FUNCTION_BLOCK "LMQTT_Client"
{ S7_Optimized_Access := 'TRUE' }
AUTHOR : 'Siemens Industry Online Support'
FAMILY : LMQTT
VERSION : 4.0
   VAR_INPUT
      enable : Bool;
      publish : Bool;
      subscribe : Bool;
      unsubscribe : Bool;
      qos : USInt;
      "retain" : Bool;
      publishMsgLen : UDInt := 0;
      willMsgLen : UInt := 0;
      timeOut { S7_HiddenAssignment := 'HideIfNoParamAssigned'} : Time := T#5s;
   END_VAR

   VAR_OUTPUT
      valid { ExternalWritable := 'False'} : Bool;
      done { ExternalWritable := 'False'} : Bool;
      busy { ExternalWritable := 'False'} : Bool;
      error { ExternalWritable := 'False'} : Bool;
      status { ExternalWritable := 'False'} : Word := #STATUS_NO_CALL;
      diagnostics { ExternalWritable := 'False'} : "typeDiagnostics";
      receivedMsgStatus { ExternalWritable := 'False'} : USInt;
      receivedMsgDataLen { ExternalWritable := 'False'} : UDInt;
   END_VAR

   VAR_IN_OUT
      connParam : "LMQTT_typeConnParam";
      clientIdentifier : WString;
      username : WString;
      password : WString;
      willtopic : WString;
      willMsgPayload : Array[*] of Byte;
      mqttTopic : WString;
      publishMsgPayload : Array[*] of Byte;
      receivedTopic : WString;
      receivedMsgPayload : Array[*] of Byte;
   END_VAR

   VAR
      statEnableOld { ExternalAccessible := 'False'; ExternalVisible := 'False'; ExternalWritable := 'False'} : Bool;
      statValid { ExternalAccessible := 'False'; ExternalVisible := 'False'; ExternalWritable := 'False'} : Bool;
      statBusy { ExternalAccessible := 'False'; ExternalVisible := 'False'; ExternalWritable := 'False'} : Bool;
      statError { ExternalAccessible := 'False'; ExternalVisible := 'False'; ExternalWritable := 'False'} : Bool;
      statErrorUserCleared { ExternalAccessible := 'False'; ExternalVisible := 'False'; ExternalWritable := 'False'} : Bool;
      statErrorAutoCleared { ExternalAccessible := 'False'; ExternalVisible := 'False'; ExternalWritable := 'False'} : Bool;
      statStatus { ExternalAccessible := 'False'; ExternalVisible := 'False'; ExternalWritable := 'False'} : Word := #STATUS_NO_CALL;
      statDone { ExternalAccessible := 'False'; ExternalVisible := 'False'; ExternalWritable := 'False'} : Bool;
      statRcvMsgStatus { ExternalAccessible := 'False'; ExternalVisible := 'False'; ExternalWritable := 'False'} : USInt;
      statRcvMsgDataLen { ExternalAccessible := 'False'; ExternalVisible := 'False'; ExternalWritable := 'False'} : UDInt;
      statSubfunctionStatus { ExternalAccessible := 'False'; ExternalVisible := 'False'; ExternalWritable := 'False'} : Word;
      statFBErrorState { ExternalAccessible := 'False'; ExternalVisible := 'False'; ExternalWritable := 'False'} : DInt;
      statFBState { ExternalAccessible := 'False'; ExternalVisible := 'False'; ExternalWritable := 'False'} : DInt := #FB_STATE_NO_PROCESSING;
      statMqttConnectState { ExternalAccessible := 'False'; ExternalVisible := 'False'; ExternalWritable := 'False'} : DInt := #MQTT_CONNECT_STATE_NO_PROCESSING;
      statMqttCommandState { ExternalAccessible := 'False'; ExternalVisible := 'False'; ExternalWritable := 'False'} : DInt := #MQTT_COMMAND_STATE_NO_PROCESSING;
      statDisablingCompleted { ExternalAccessible := 'False'; ExternalVisible := 'False'; ExternalWritable := 'False'} : Bool;
      statEmptyDiagnostics { ExternalAccessible := 'False'; ExternalVisible := 'False'; ExternalWritable := 'False'; S7_SetPoint := 'False'} : "typeDiagnostics";
      statConnParam { ExternalAccessible := 'False'; ExternalVisible := 'False'; ExternalWritable := 'False'} : Struct
         isQDN { ExternalAccessible := 'False'; ExternalVisible := 'False'; ExternalWritable := 'False'} : Bool;
         paramQDN {InstructionName := 'TCON_QDN_SEC'; LibVersion := '1.0'; ExternalAccessible := 'False'; ExternalVisible := 'False'; ExternalWritable := 'False'; S7_SetPoint := 'False'} : TCON_QDN_SEC;
         paramIP {InstructionName := 'TCON_IP_V4_SEC'; LibVersion := '1.0'; ExternalAccessible := 'False'; ExternalVisible := 'False'; ExternalWritable := 'False'; S7_SetPoint := 'False'} : TCON_IP_V4_SEC;
      END_STRUCT;
      instTsendC {InstructionName := 'TSEND_C'; LibVersion := '3.2'; ExternalAccessible := 'False'; ExternalVisible := 'False'; ExternalWritable := 'False'; S7_SetPoint := 'False'} : TSEND_C;
      instTrcv {InstructionName := 'TRCV'; LibVersion := '4.0'; ExternalAccessible := 'False'; ExternalVisible := 'False'; ExternalWritable := 'False'; S7_SetPoint := 'False'} : TRCV;
      statSendBuffer { ExternalAccessible := 'False'; ExternalVisible := 'False'; ExternalWritable := 'False'} : Array[0..#MAX_BUFFER_LEN_SEND] of Byte;
      statRcvBuffer { ExternalAccessible := 'False'; ExternalVisible := 'False'; ExternalWritable := 'False'} : Array[0..#MAX_BUFFER_LEN_RCV] of Byte;
      statPublishOld { ExternalAccessible := 'False'; ExternalVisible := 'False'; ExternalWritable := 'False'} : Bool;
      statSubscribeOld { ExternalAccessible := 'False'; ExternalVisible := 'False'; ExternalWritable := 'False'} : Bool;
      statUnsubscribeOld { ExternalAccessible := 'False'; ExternalVisible := 'False'; ExternalWritable := 'False'} : Bool;
      statTsendcReq { ExternalAccessible := 'False'; ExternalVisible := 'False'; ExternalWritable := 'False'} : Bool;
      statTsendcEnable { ExternalAccessible := 'False'; ExternalVisible := 'False'; ExternalWritable := 'False'} : Bool;
      statTsendcLen { ExternalAccessible := 'False'; ExternalVisible := 'False'; ExternalWritable := 'False'} : UDInt;
      statEnableTimerCommandWatchdog { ExternalAccessible := 'False'; ExternalVisible := 'False'; ExternalWritable := 'False'} : Bool;
      instTimerCommandWatchdog {InstructionName := 'IEC_TIMER'; LibVersion := '1.0'; ExternalAccessible := 'False'; ExternalVisible := 'False'; ExternalWritable := 'False'; S7_SetPoint := 'False'} : IEC_TIMER;
      statEnableMqttKeepAliveTimer { ExternalAccessible := 'False'; ExternalVisible := 'False'; ExternalWritable := 'False'} : Bool;
      statMqttKeepAliveUsed { ExternalAccessible := 'False'; ExternalVisible := 'False'; ExternalWritable := 'False'} : Bool;
      statMqttKeepAliveTime { ExternalAccessible := 'False'; ExternalVisible := 'False'; ExternalWritable := 'False'} : Time;
      instMqttKeepAliveTimer {InstructionName := 'IEC_TIMER'; LibVersion := '1.0'; ExternalAccessible := 'False'; ExternalVisible := 'False'; ExternalWritable := 'False'; S7_SetPoint := 'False'} : IEC_TIMER;
      statSendBufferPos { ExternalAccessible := 'False'; ExternalVisible := 'False'; ExternalWritable := 'False'} : UInt;
      statPaketHeaderEncodeDone { ExternalAccessible := 'False'; ExternalVisible := 'False'; ExternalWritable := 'False'} : Bool;
      statSendPaketTotalRemLen { ExternalAccessible := 'False'; ExternalVisible := 'False'; ExternalWritable := 'False'} : UDInt;
      statEncodedRemPaketLenAsByte { ExternalAccessible := 'False'; ExternalVisible := 'False'; ExternalWritable := 'False'} : Byte;
      statUsernameLenUtf8Encoded { ExternalAccessible := 'False'; ExternalVisible := 'False'; ExternalWritable := 'False'} : UInt;
      statPasswordLenUtf8Encoded { ExternalAccessible := 'False'; ExternalVisible := 'False'; ExternalWritable := 'False'} : UInt;
      statWillTopicLenUtf8Encoded { ExternalAccessible := 'False'; ExternalVisible := 'False'; ExternalWritable := 'False'} : UInt;
      statClientIdLenUtf8Encoded { ExternalAccessible := 'False'; ExternalVisible := 'False'; ExternalWritable := 'False'} : UInt;
      statWillQos { ExternalAccessible := 'False'; ExternalVisible := 'False'; ExternalWritable := 'False'} : USInt;
      statWillRetain { ExternalAccessible := 'False'; ExternalVisible := 'False'; ExternalWritable := 'False'} : Bool;
      statWillMessageCnt { ExternalAccessible := 'False'; ExternalVisible := 'False'; ExternalWritable := 'False'} : UInt;
      statClientIdPos { ExternalAccessible := 'False'; ExternalVisible := 'False'; ExternalWritable := 'False'} : DInt;
      statClientIdEncodeState { ExternalAccessible := 'False'; ExternalVisible := 'False'; ExternalWritable := 'False'} : DInt;
      statWillMessagePos { ExternalAccessible := 'False'; ExternalVisible := 'False'; ExternalWritable := 'False'} : DInt;
      statWillMessageEncodeState { ExternalAccessible := 'False'; ExternalVisible := 'False'; ExternalWritable := 'False'} : DInt;
      statWillTopicPos { ExternalAccessible := 'False'; ExternalVisible := 'False'; ExternalWritable := 'False'} : DInt;
      statWillTopicEncodeState { ExternalAccessible := 'False'; ExternalVisible := 'False'; ExternalWritable := 'False'} : DInt;
      statUserNamePos { ExternalAccessible := 'False'; ExternalVisible := 'False'; ExternalWritable := 'False'} : DInt;
      statUserNameEncodeState { ExternalAccessible := 'False'; ExternalVisible := 'False'; ExternalWritable := 'False'} : DInt;
      statPasswordPos { ExternalAccessible := 'False'; ExternalVisible := 'False'; ExternalWritable := 'False'} : DInt;
      statPasswordEncodeState { ExternalAccessible := 'False'; ExternalVisible := 'False'; ExternalWritable := 'False'} : DInt;
      statPaketId { ExternalAccessible := 'False'; ExternalVisible := 'False'; ExternalWritable := 'False'} : UInt;
      statPublishTopicLenUtf8Encoded { ExternalAccessible := 'False'; ExternalVisible := 'False'; ExternalWritable := 'False'} : UInt;
      statPublishQos { ExternalAccessible := 'False'; ExternalVisible := 'False'; ExternalWritable := 'False'} : USInt;
      statPublishMessageCnt { ExternalAccessible := 'False'; ExternalVisible := 'False'; ExternalWritable := 'False'} : UDInt;
      statPublishTopicEncodeState { ExternalAccessible := 'False'; ExternalVisible := 'False'; ExternalWritable := 'False'} : DInt;
      statPublishTopicPos { ExternalAccessible := 'False'; ExternalVisible := 'False'; ExternalWritable := 'False'} : DInt;
      statPaketIdEncoded { ExternalAccessible := 'False'; ExternalVisible := 'False'; ExternalWritable := 'False'} : Bool;
      statPublishEncodeMessageState { ExternalAccessible := 'False'; ExternalVisible := 'False'; ExternalWritable := 'False'} : DInt;
      statPublishMessagePos { ExternalAccessible := 'False'; ExternalVisible := 'False'; ExternalWritable := 'False'} : DInt;
      statSubscribeQos { ExternalAccessible := 'False'; ExternalVisible := 'False'; ExternalWritable := 'False'} : USInt;
      statSubscribeQosEncoded { ExternalAccessible := 'False'; ExternalVisible := 'False'; ExternalWritable := 'False'} : Bool;
      statSubscribeTopicPos { ExternalAccessible := 'False'; ExternalVisible := 'False'; ExternalWritable := 'False'} : DInt;
      statSubscribeTopicEncodeState { ExternalAccessible := 'False'; ExternalVisible := 'False'; ExternalWritable := 'False'} : DInt;
      statSubscribeTopicLenUtf8Encoded { ExternalAccessible := 'False'; ExternalVisible := 'False'; ExternalWritable := 'False'} : UInt;
      statUnsubscribeTopicPos { ExternalAccessible := 'False'; ExternalVisible := 'False'; ExternalWritable := 'False'} : DInt;
      statUnsubscribeTopicEncodeState { ExternalAccessible := 'False'; ExternalVisible := 'False'; ExternalWritable := 'False'} : DInt;
      statUnsubscribeTopicLenUtf8Encoded { ExternalAccessible := 'False'; ExternalVisible := 'False'; ExternalWritable := 'False'} : UInt;
      statRcvMsgQoS { ExternalAccessible := 'False'; ExternalVisible := 'False'; ExternalWritable := 'False'} : UInt;
      statRcvMsgTotalLen { ExternalAccessible := 'False'; ExternalVisible := 'False'; ExternalWritable := 'False'} : UDInt;
      statRcvMsgTopicLen { ExternalAccessible := 'False'; ExternalVisible := 'False'; ExternalWritable := 'False'} : UInt;
      statRcvMsgPayloadLen { ExternalAccessible := 'False'; ExternalVisible := 'False'; ExternalWritable := 'False'} : UDInt;
      statRcvMsgPaketId { ExternalAccessible := 'False'; ExternalVisible := 'False'; ExternalWritable := 'False'} : Word;
      statRcvMsgTopicPos { ExternalAccessible := 'False'; ExternalVisible := 'False'; ExternalWritable := 'False'} : DInt;
      statRcvMsgPayloadPos { ExternalAccessible := 'False'; ExternalVisible := 'False'; ExternalWritable := 'False'} : DInt;
      statRcvMsgDecodeState { ExternalAccessible := 'False'; ExternalVisible := 'False'; ExternalWritable := 'False'} : DInt;
      statRcvMsgInternalStatus { ExternalAccessible := 'False'; ExternalVisible := 'False'; ExternalWritable := 'False'} : USInt;
      statMqttPubRecRcv { ExternalAccessible := 'False'; ExternalVisible := 'False'; ExternalWritable := 'False'} : USInt;
      statSendPubAckMsg { ExternalAccessible := 'False'; ExternalVisible := 'False'; ExternalWritable := 'False'} : Bool;
      statPubRecReady { ExternalAccessible := 'False'; ExternalVisible := 'False'; ExternalWritable := 'False'} : Bool;
      statCommandInputOld { ExternalAccessible := 'False'; ExternalVisible := 'False'; ExternalWritable := 'False'} : Bool;
      statCommandInputBackup { ExternalAccessible := 'False'; ExternalVisible := 'False'; ExternalWritable := 'False'} : Byte;
   END_VAR

   VAR_TEMP
      tempEnable : Bool;
      tempSubscribe : Bool;
      tempPublish : Bool;
      tempUnsubscribe : Bool;
      tempTsendcDone : Bool;
      tempTsendcBusy : Bool;
      tempTsendcError : Bool;
      tempTsendcStatus : Word;
      tempTrcvNdr : Bool;
      tempTrcvBusy : Bool;
      tempTrcvError : Bool;
      tempTrcvStatus : Word;
      tempTrcvRcvdLen : UDInt;
      tempTrcvBufferPos : DInt;
      tempUserFlag : Bool;
      tempPasswordFlag : Bool;
      tempWillFlag : Bool;
      tempWillQoS1 : Bool;
      tempWillQoS2 : Bool;
      tempMaxWillMsgLen : DInt;
      tempLowerWillMsgArrayBoundary : DInt;
      tempLoopCounter : DInt;
      tempBytesUsedUtf8 : USInt;
      tempErrorConvertUtf8 : Bool;
      tempStatusConvertUtf8 : Word;
      tempConvertedUtf8 : DWord;
      tempWordForSliceAddress : Word;
      tempCommandInput : Byte;
      tempRcvMsgTypeCase : Byte;
      tempMaxPublishDataArrayLen : DInt;
      tempMqttConnAckRcvStatus : USInt;
      tempMqttPingRspRcv : USInt;
      tempMqttPubAckRcv : USInt;
      tempMqttPubCompRcv : USInt;
      tempMqttSubAckRcv : USInt;
      tempMqttUnSubAckRcv : USInt;
      tempLowerBoundPublishDataArray : DInt;
      tempMultiplierToDecode : UDInt;
      tempReceivedTopicStringMaxLen : DInt;
      tempReceivedMsgDataArrayTotalLen : DInt;
      tempUpperBoundRcvMsgDataArray : DInt;
      tempFirstChar : Int;
   END_VAR

   VAR CONSTANT
      FB_STATE_NO_PROCESSING : DInt := 0;
      FB_STATE_VALIDATE_INPUT : DInt := 10;
      FB_STATE_TCP_CONNECTING : DInt := 20;
      FB_STATE_OPERATING_MONITOR_TCP : DInt := 30;
      FB_STATE_TCP_RECONNECTING : DInt := 40;
      FB_STATE_DISABLING : DInt := 90;
      MQTT_CONNECT_STATE_NO_PROCESSING : DInt := 0;
      MQTT_CONNECT_STATE_BUILD_PAKET : DInt := 100;
      MQTT_CONNECT_STATE_SEND_PAKET_WAIT_FOR_CONNACK : DInt := 200;
      MQTT_CONNECT_STATE_CONNECTED : DInt := 300;
      MQTT_CONNECT_STATE_DISCONNECTED : DInt := 400;
      MQTT_COMMAND_STATE_NO_PROCESSING : DInt := 0;
      MQTT_COMMAND_STATE_BUILD_PUBLISH : DInt := 1;
      MQTT_COMMAND_STATE_SEND_PUBLISH : DInt := 1000;
      MQTT_COMMAND_STATE_BUILD_SUBSCRIBE : DInt := 2;
      MQTT_COMMAND_STATE_SEND_SUBSCRIBE : DInt := 2000;
      MQTT_COMMAND_STATE_BUILD_UNSUBSCRIBE : DInt := 4;
      MQTT_COMMAND_STATE_SEND_UNSUBSCRIBE : DInt := 3000;
      MQTT_COMMAND_STATE_SEND_PING : DInt := 8000;
      MQTT_COMMAND_STATE_PING_RESP : DInt := 9000;
      STATUS_JOB_EXECUTED : Word := 16#0000;
      STATUS_NO_CALL : Word := 16#7000;
      STATUS_FIRST_CALL : Word := 16#7001;
      STATUS_SUBSEQUENT_CALL : Word := 16#7002;
      STATUS_MQTT_CONNECTING : Word := 16#7003;
      STATUS_MQTT_CONNECTED : Word := 16#7004;
      STATUS_MQTT_PING : Word := 16#7005;
      STATUS_MQTT_PUBLISH : Word := 16#7006;
      STATUS_MQTT_SUBSCRIBE : Word := 16#7008;
      STATUS_MQTT_UNSUBSCRIBE : Word := 16#7010;
      ERR_UNDEFINED_STATE : Word := 16#8600;
      ERR_TCP_RECONNECTING : Word := 16#9000;
      ERR_CLIENT_ID_NULL : Word := 16#8200;
      ERR_BROKER_INVALID : Word := 16#8201;
      ERR_CNT_EXCEEDS_ARRAY_DIMENSION : Word := 16#8210;
      ERR_KEEPALIVE_INVALID : Word := 16#8220;
      ERR_QOS_INVALID : Word := 16#8230;
      ERR_TCON_FAILED : Word := 16#8601;
      ERR_TCON_TIMEOUT : Word := 16#8620;
      ERR_MQTT_REM_LEN_INVALID : Word := 16#8700;
      ERR_MQTT_MALFORMED_QOS_RECEIVED : Word := 16#8710;
      ERR_MQTT_CONNACK_INVALID_SESSION_FLAG : Word := 16#8720;
      ERR_MQTT_CONNACK_RETURN_CODE_INVALID : Word := 16#8730;
      ERR_MQTT_PAKET_ID_INVALID : Word := 16#8740;
      ERR_MQTT_SUBACK_FAILURE : Word := 16#8750;
      ERR_MQTT_COMMAND_MULTIPLE_INPUT : Word := 16#8001;
      ERR_MQTT_COMMAND_PUBLISH_TOPIC_INVALID : Word := 16#8300;
      ERR_MQTT_COMMAND_SUBSCRIBE_TOPIC_INVALID : Word := 16#8310;
      ERR_MQTT_COMMAND_UNSUBSCRIBE_TOPIC_INVALID : Word := 16#8320;
      ERR_MQTT_COMMAND_SEND_TIMEOUT : Word := 16#8650;
      ERR_MQTT_CONNECT_TIMEOUT : Word := 16#8670;
      MAX_BUFFER_LEN_RCV : UInt := 1459;
      MAX_BUFFER_LEN_SEND : UInt := 8191;
      EMPTY_BYTE : Byte := 16#00;
      NO_COMMAND : Byte := 16#00;
      EMPTY_STRING : String;
      EMPTY_WSTRING : WString;
      LEN_NULL : Int := 0;
      INIT_UDINT_1 : UDInt := 1;
      ARRAY_LEN_OFFSET_PLUS_1 : DInt := 1;
      FIRST_CHARACTER : DInt := 1;
      ONE_DIMENSION : UDInt := 1;
      FIRST_ENCODING : DInt := 1;
      SUBSEQUENT_ENCODING : DInt := 2;
      ENCODE_DONE : DInt := 3;
      NOT_USED_NO_ENCODING : DInt := 5;
      MSG_DECODE_STATE_NO_PROCESSING : DInt := 0;
      MSG_DECODE_STATE_TOPIC : DInt := 1;
      MSG_DECODE_STATE_PAKET_ID_MSB : DInt := 2;
      MSG_DECODE_STATE_PAKET_ID_LSB : DInt := 3;
      MSG_DECODE_STATE_PAYLOAD : DInt := 4;
      MSG_DECODE_STATUS_NO_NEW_MSG : USInt := 0;
      MSG_DECODE_STATUS_NEW_MSG_OK : USInt := 1;
      MSG_DECODE_STATUS_TOPIC_TOO_LONG : USInt := 2;
      MSG_DECODE_STATUS_PAYLOAD_TOO_LONG : USInt := 2;
      MQTT_QOS_0 : UInt := 0;
      MQTT_QOS_1 : UInt := 1;
      MQTT_QOS_2 : UInt := 2;
      REMAINING_LEN_3 : Byte := 16#03;
      REMAINING_LEN_2 : Byte := 16#02;
      REMAINIG_LEN_0 : Byte := 16#00;
      SUBSCRIBE_FAILURE : Byte := 16#80;
      MQTT_NO_SESSION_PRESENT : Byte := 16#00;
      KEEPALIVE_DISABLED : Time := t#0s;
      TSENDC_JOB_DONE : Word := 16#0000;
      TSENDC_COM_CLOSED : Word := 16#0003;
      TSENDC_EST_OK : Word := 16#7004;
      TSENDC_DISCONNECTED : Word := 16#7000;
      UINT_CONST_1000 : UInt := 1000;
      TWO_SECONDS : UInt := 2000;
      THREE_SECONDS : UInt := 3;
      UTF_1_BYTE_USED : USInt := 1;
      UTF_2_BYTE_USED : USInt := 2;
      UTF_3_BYTE_USED : USInt := 3;
      ONE_BYTE_LEN_INFO : UInt := 1;
      TWO_BYTE_LEN_INFO : UInt := 2;
      CONNECT_HEADER_10BYTE_LEN : UInt := 10;
      NO_RESPONSE : USInt := 0;
      RESPONSE_GOOD : USInt := 1;
      RESPONSE_PAKET_ID_INVALID : USInt := 2;
      RESPONSE_SUBSCRIBE_FAILED : USInt := 3;
      MQTT_MSG_TYPE_CONNECT : Byte := 16#10;
      MQTT_MSG_TYPE_CONNACK : Byte := 16#20;
      MQTT_MSG_TYPE_DISCONNECT : Byte := 16#E0;
      MQTT_MSG_TYPE_PUBLISH : Byte := 16#30;
      MQTT_MSG_TYPE_PUBACK : Byte := 16#40;
      MQTT_MSG_TYPE_PUBREC : Byte := 16#50;
      MQTT_MSG_TYPE_PUBREL : Byte := 16#62;
      MQTT_MSG_TYPE_PUBCOMP : Byte := 16#70;
      MQTT_MSG_TYPE_SUBSCRIBE : Byte := 16#82;
      MQTT_MSG_TYPE_UNSUBSCRIBE : Byte := 16#A2;
      MQTT_MSG_TYPE_SUBACK : Byte := 16#90;
      MQTT_MSG_TYPE_UNSUBACK : Byte := 16#B0;
      MQTT_MSG_TYPE_PING : Byte := 16#C0;
      MQTT_MSG_TYPE_PINGRESP : Byte := 16#D0;
      MQTT_MSG_TYPE_RCV_PUB_MESSAGE : Byte := 16#30;
      MQTT_MSG_TYPE_RCV_PUB_MESSAGE_QoS0 : Byte := 16#30;
      MQTT_MSG_TYPE_RCV_PUB_MESSAGE_QoS1 : Byte := 16#32;
      MQTT_MSG_TYPE_RCV_PUB_MESSAGE_QoS2 : Byte := 16#34;
      MQTT_MSG_TYPE_RCV_PUB_MESSAGE_BAD : Byte := 16#36;
      MQTT_MSG_DECODING : Byte := 16#FF;
      MQTT_CONNACK_ACCEPTED : Byte := 16#00;
      BIT_MASK_HIGHBITS : Byte := 16#F0;
      BIT_MASK_QOS : Byte := 16#F6;
      DEFAULT_VALUE_ZERO : Int := 0;
      SEND_LEN_MULTIPLIER_UDINT_128 : UDInt := 128;
      MAX_ALLOWED_PAKET_SIZE : UDInt := 2097152;
      DEFAULT_MULTIPLIER_BYTE_127 : Byte := 16#7F;
      CONN_PROTOCOL_NAME_0 : Byte := 16#00;
      CONN_PROTOCOL_NAME_4 : Byte := 16#04;
      CONN_PROTOCOL_MQTT_VERSION_3_1_1 : Byte := 16#04;
   END_VAR


BEGIN
	REGION BLOCK INFO HEADER
	  //===============================================================================
	  // SIEMENS (c)Copyright 2023
	  //-------------------------------------------------------------------------------
	  // Title:        LMQTT_Client
	  // Function:     This FB implements an MQTT client. A user can publish data and
	  //               subscribe to topics to receive data.
	  // Library:      LMQTT
	  // Author:       Siemens Industry Online Support
	  // Tested with:  CPU 1516-3 PN/DP FW 2.9
	  // Engineering:  TIA Portal V17
	  // Restrictions: --
	  // Requirements: S7-1200 with firmware V4.4 or higher
	  //               S7-1500 with firmware V2.0 or higher
	  //-------------------------------------------------------------------------------
	  // Change log table:
	  // Version  | Date       | Expert in charge       | Changes applied
	  //----------|------------|------------------------|------------------------------
	  // 04.00.03 | 2024-04-09 | Online Support         | Allowed lastWill without payload
	  // 04.00.03 | 2024-02-12 | Online Support         | Improved evaluation of broker address
	  // 04.00.02 | 2023-09-05 | Online Support         | Fixed bug that edge on publish/subscribe while PING is saved
	  // 04.00.01 | 2023-08-30 | Online Support         | Fixed bug at TRCV and ConnID
	  // 04.00.00 | 2023-08-04 | Online Support         | Broker can be addresses with hostname or IP address using one parameter
	  //                                                | Reordered interface
	  //                                                | Fixed bug at publish with QoS = 2
	  // 03.00.05 | 2023-02-23 | Online Support         | Fixed bug that in rare situations no new commands were accepted
	  // 03.00.04 | 2022-06-09 | Online Support         | Fixed bug that done was not set if input was reset
	  // 03.00.03 | 2021-05-07 | Online Support         | Minor bug fixes
	  // 03.00.00 | 2020-11-04 | Online Support         | New block interface with major improvements
	  // 02.02.02 | 2020-03-16 | Online Support         | Improved issue with validateSubjectAlternateNameOfServer not setting correct bit
	  // 02.02.01 | 2019-12-03 | Online Support         | Update to V16 and fusion with S7-1200 Lib
	  // 02.01.00 | 2019-11-10 | Online Support         | Minor connection improvements. Updated some comments
	  // 02.00.00 | 2018-06-04 | Online Support         | Added DNS support and Subscribe to topics
	  // 01.00.00 | 2017-06-06 | Online Support         | First released version
	  //===============================================================================
	END_REGION

	#tempEnable := #enable; // Work with temporary value / create process image
	#tempPublish := #publish;  // Work with temporary value / create process image - only checked when MQTT is connected
	#tempSubscribe := #subscribe;  // Work with temporary value / create process image - only checked when MQTT is connected
	#tempUnsubscribe := #unsubscribe;  // Work with temporary value / create process image - only checked when MQTT is connected


	REGION OUC_BLOCK_CALLS
	  //Only call if FB is processing
	  IF #statStatus <> #STATUS_NO_CALL THEN
	    // Connect and send
	    IF #statConnParam.isQDN = TRUE THEN // Call if host is a domain name
	      #instTsendC(REQ     := #statTsendcReq,
	                  CONT    := #statTsendcEnable,
	                  LEN     := #statTsendcLen,
	                  DONE    => #tempTsendcDone,
	                  BUSY    => #tempTsendcBusy,
	                  ERROR   => #tempTsendcError,
	                  STATUS  => #tempTsendcStatus,
	                  CONNECT := #statConnParam.paramQDN,
	                  DATA    := #statSendBuffer);

	    ELSE
	      #instTsendC(REQ     := #statTsendcReq,
	                  CONT    := #statTsendcEnable,
	                  LEN     := #statTsendcLen,
	                  DONE    => #tempTsendcDone,
	                  BUSY    => #tempTsendcBusy,
	                  ERROR   => #tempTsendcError,
	                  STATUS  => #tempTsendcStatus,
	                  CONNECT := #statConnParam.paramIP,
	                  DATA    := #statSendBuffer);
	    END_IF;

	    // Receive only when TCP operating
	    #instTrcv(EN_R     := (#statFBState = #FB_STATE_OPERATING_MONITOR_TCP),
	              ID       := #statConnParam.paramQDN.ConnPara.ID,
	              ADHOC    := true,
	              NDR      => #tempTrcvNdr,
	              BUSY     => #tempTrcvBusy,
	              ERROR    => #tempTrcvError,
	              STATUS   => #tempTrcvStatus,
	              RCVD_LEN => #tempTrcvRcvdLen,
	              DATA     := #statRcvBuffer);

	    //Monitor Time out
	    #instTimerCommandWatchdog.TON(IN := #statEnableTimerCommandWatchdog,
	                                  PT := #timeOut);
	    //Mqtt Keepalive Timer
	    #instMqttKeepAliveTimer.TON(IN := #statEnableMqttKeepAliveTimer,
	                                PT := #statMqttKeepAliveTime);
	  END_IF;
	END_REGION

	REGION ENABLING/DISABLING_FUNCTION_BLOCK
	  IF (#tempEnable = TRUE) AND (#statStatus = #STATUS_NO_CALL) THEN // Enable FB
	    // First call; initialize FB
	    #statValid := TRUE;
	    #statBusy := TRUE;
	    #statError := FALSE;
	    #statDone := FALSE;
	    #statErrorUserCleared := FALSE;
	    #statErrorAutoCleared := FALSE;
	    #statStatus := #STATUS_FIRST_CALL;
	    #statSubfunctionStatus := #STATUS_JOB_EXECUTED;
	    #statFBErrorState := 0;
	    #diagnostics := #statEmptyDiagnostics;
	    #statDisablingCompleted := FALSE;
	    // State machine - start functionality
	    #statFBState := #FB_STATE_VALIDATE_INPUT;

	    // Initialize functionality: reset of variables, diagnostics, etc.
	    #statPublishOld := FALSE;
	    #statSubscribeOld := FALSE;
	    #statUnsubscribeOld := FALSE;
	    #statConnParam.isQDN := FALSE;
	    #statTsendcReq := FALSE;
	    #statTsendcEnable := FALSE;
	    #statTsendcLen := 0;
	    #statEnableTimerCommandWatchdog := FALSE;
	    #statEnableMqttKeepAliveTimer := FALSE;
	    #statMqttKeepAliveTime := #KEEPALIVE_DISABLED;
	    #statMqttKeepAliveUsed := FALSE;
	    #statSendBufferPos := 0;
	    #statPaketHeaderEncodeDone := FALSE;
	    #statSendPaketTotalRemLen := 0;
	    #statEncodedRemPaketLenAsByte := #EMPTY_BYTE;
	    #statClientIdPos := 0;
	    #statClientIdEncodeState := 0;
	    #statClientIdLenUtf8Encoded := 0;
	    #statUserNamePos := 0;
	    #statUserNameEncodeState := #FIRST_ENCODING;
	    #statUsernameLenUtf8Encoded := 0;
	    #statPasswordPos := 0;
	    #statPasswordEncodeState := #FIRST_ENCODING;
	    #statPasswordLenUtf8Encoded := 0;
	    #statWillQos := 0;
	    #statWillRetain := FALSE;
	    #statWillMessageCnt := 0;
	    #statWillMessagePos := 0;
	    #statWillMessageEncodeState := #FIRST_ENCODING;
	    #statWillTopicLenUtf8Encoded := 0;
	    #statWillTopicPos := 0;
	    #statWillTopicEncodeState := #FIRST_ENCODING;
	    #statPaketId := 0;
	    #statPublishTopicLenUtf8Encoded := 0;
	    #statPublishQos := 0;
	    #statPublishMessageCnt := 0;
	    #statPublishTopicEncodeState := #FIRST_ENCODING;
	    #statPublishTopicPos := 0;
	    #statPaketIdEncoded := FALSE;
	    #statPublishEncodeMessageState := #FIRST_ENCODING;
	    #statPublishMessagePos := 0;
	    #statSubscribeQos := 0;
	    #statSubscribeQosEncoded := FALSE;
	    #statSubscribeTopicPos := 0;
	    #statSubscribeTopicEncodeState := #FIRST_ENCODING;
	    #statSubscribeTopicLenUtf8Encoded := 0;
	    #statUnsubscribeTopicPos := 0;
	    #statUnsubscribeTopicEncodeState := #FIRST_ENCODING;
	    #statUnsubscribeTopicLenUtf8Encoded := 0;
	    #statRcvMsgQoS := 0;
	    #statRcvMsgTotalLen := 0;
	    #statRcvMsgTopicLen := 0;
	    #statRcvMsgPayloadLen := 0;
	    #statRcvMsgPaketId := 0;
	    #statRcvMsgTopicPos := 0;
	    #statRcvMsgPayloadPos := 0;
	    #statRcvMsgDecodeState := #MSG_DECODE_STATE_NO_PROCESSING;
	    #statRcvMsgInternalStatus := 0;
	    #statRcvMsgStatus := 0;
	    #statRcvMsgDataLen := 0;
	    #statSendPubAckMsg := FALSE;

	    // Initialize functionality: call subsidiary FBs with FALSE
	    FILL_BLK(IN    := #EMPTY_BYTE,
	             COUNT := #MAX_BUFFER_LEN_SEND,
	             OUT   => #statSendBuffer[0]);
	    FILL_BLK(IN    := #EMPTY_BYTE,
	             COUNT := #MAX_BUFFER_LEN_RCV,
	             OUT   => #statRcvBuffer[0]);
	    RESET_TIMER(#instTimerCommandWatchdog);
	    RESET_TIMER(#instMqttKeepAliveTimer);

	    // INIT SUB STATE MACHINES
	    #statMqttConnectState := #MQTT_CONNECT_STATE_NO_PROCESSING;
	    #statMqttCommandState := #MQTT_COMMAND_STATE_NO_PROCESSING;
	    #statRcvMsgDecodeState := #MSG_DECODE_STATE_NO_PROCESSING;

	  ELSIF (#tempEnable = FALSE) AND (#statEnableOld = TRUE) THEN // Disable FB
	    #statFBState := #FB_STATE_DISABLING;
	  ELSIF (#statStatus = #STATUS_FIRST_CALL) THEN // Set status identifier of subsequent call
	    #statStatus := #STATUS_SUBSEQUENT_CALL;
	  END_IF;

	  // Edge detection 'enable' input
	  #statEnableOld := #tempEnable;
	END_REGION ENABLING/DISABLING

	IF (#statStatus = #STATUS_NO_CALL) THEN // Nothing to do -> End here to reduce "system load"
	  RETURN;
	END_IF;

	REGION STATE_MACHINE_FUNCTION_BLOCK_TCP
	  CASE #statFBState OF // State machine of FB
	    #FB_STATE_NO_PROCESSING: // No processing active (Note: this state must always be present and left empty)
	      ;

	    #FB_STATE_VALIDATE_INPUT: // Enabling active
	      REGION EVALUATE CONNECTION PARAMETERS
	        // Determine if host is domain name or IP address
	        #statConnParam.isQDN := NOT "IsIPAddress"(address := #connParam.broker, ipAddress => #statConnParam.paramIP.ConnPara.RemoteAddress);

	        IF #statConnParam.isQDN THEN // Broker address is a hostname
	          IF #connParam.broker[LEN(#connParam.broker)] = '.' THEN
	            #statConnParam.paramQDN.ConnPara.RemoteQDN := #connParam.broker;
	          ELSE
	            #statConnParam.paramQDN.ConnPara.RemoteQDN := CONCAT(IN1 := #connParam.broker, IN2 := '.');
	          END_IF;

	          #statConnParam.paramQDN.ConnPara.InterfaceId := #connParam.hwId;
	          #statConnParam.paramQDN.ConnPara.ID := #connParam.connId;
	          #statConnParam.paramQDN.ConnPara.ActiveEstablished := TRUE;
	          #statConnParam.paramQDN.ConnPara.RemotePort := #connParam."port";
	        ELSE // Broker address is an IP address
	          #statConnParam.paramIP.ConnPara.InterfaceId := #connParam.hwId;
	          #statConnParam.paramIP.ConnPara.ID := #statConnParam.paramQDN.ConnPara.ID := #connParam.connId;
	          #statConnParam.paramIP.ConnPara.ActiveEstablished := TRUE;
	          #statConnParam.paramIP.ConnPara.RemotePort := #connParam."port";
	        END_IF;

	        IF #connParam.tls.enableTls THEN
	          IF #statConnParam.isQDN THEN
	            #statConnParam.paramQDN.ActivateSecureConn := TRUE;
	            #statConnParam.paramQDN.ExtTLSCapabilities.%X0 := #connParam.tls.validateServerIdentity;
	            #statConnParam.paramQDN.TLSServerCertRef := #connParam.tls.brokerCert;
	            #statConnParam.paramQDN.TLSClientCertRef := #connParam.tls.clientCert;
	          ELSE
	            #statConnParam.paramIP.ActivateSecureConn := TRUE;
	            #statConnParam.paramIP.ExtTLSCapabilities.%X0 := #connParam.tls.validateServerIdentity;
	            #statConnParam.paramIP.TLSServerCertRef := #connParam.tls.brokerCert;
	            #statConnParam.paramIP.TLSClientCertRef := #connParam.tls.clientCert;
	          END_IF;
	        END_IF;
	      END_REGION EVALUATE CONNECTION PARAMETERS

	      REGION FB_VALIDATE_INPUT
	        //Check Input variables:
	        #tempMaxWillMsgLen := ABS(UPPER_BOUND(ARR := #willMsgPayload, DIM := #ONE_DIMENSION) - LOWER_BOUND(ARR := #willMsgPayload, DIM := #ONE_DIMENSION)) + #ARRAY_LEN_OFFSET_PLUS_1;

	        //Check Client ID len Must be > 0
	        IF LEN(#clientIdentifier) <= #LEN_NULL THEN
	          #statStatus := #ERR_CLIENT_ID_NULL; // Set correct status that identifies error clearly
	          #statSubfunctionStatus := #ERR_CLIENT_ID_NULL; // Status or return value of called FBs, FCs and system blocks
	          #statFBErrorState := #statFBState; // Set error state number for diagnostic
	          #statErrorUserCleared := TRUE;
	          //verify Will next
	        ELSIF #tempMaxWillMsgLen < #willMsgLen THEN
	          #statStatus := #ERR_CNT_EXCEEDS_ARRAY_DIMENSION; // Set correct status that identifies error clearly
	          #statSubfunctionStatus := #ERR_CNT_EXCEEDS_ARRAY_DIMENSION; // Status or return value of called FBs, FCs and system blocks
	          #statFBErrorState := #statFBState; // Set error state number for diagnostic
	          #statErrorUserCleared := TRUE;
	          ///CHECK WILL QOS
	        ELSIF #qos > #MQTT_QOS_2 THEN
	          #statStatus := #ERR_QOS_INVALID; // Set correct status that identifies error clearly
	          #statSubfunctionStatus := #ERR_QOS_INVALID; // Status or return value of called FBs, FCs and system blocks
	          #statFBErrorState := #statFBState; // Set error state number for diagnostic
	          #statErrorUserCleared := TRUE;
	        ELSIF (#connParam.keepAlive < #THREE_SECONDS) // IF Set to 1 or 2 seconds..
	          AND (#connParam.keepAlive > 0)
	        THEN
	          #statStatus := #ERR_KEEPALIVE_INVALID; // Set correct status that identifies error clearly
	          #statSubfunctionStatus := #ERR_KEEPALIVE_INVALID; // Status or return value of called FBs, FCs and system blocks
	          #statFBErrorState := #statFBState; // Set error state number for diagnostic
	          #statErrorUserCleared := TRUE;
	        ELSE
	          //Set Params for connection
	          //Set Client Id
	          #statWillQos := #qos;
	          //set Retain
	          #statWillRetain := #retain;
	          // Will message cnt
	          #statWillMessageCnt := #willMsgLen;

	          //Keepalive
	          IF #connParam.keepAlive = 0 THEN
	            #statMqttKeepAliveUsed := FALSE;
	          ELSE
	            #statMqttKeepAliveUsed := TRUE;
	            //KeepAliveTImer is set to ((Keep Alive converted to seconds) - 2s)
	            #statMqttKeepAliveTime := UINT_TO_TIME((#connParam.keepAlive * #UINT_CONST_1000 - #TWO_SECONDS));
	          END_IF;

	          //rdy to enable TCON
	          #statTsendcEnable := TRUE;
	          #statEnableTimerCommandWatchdog := TRUE;
	          #statFBState := #FB_STATE_TCP_CONNECTING;
	        END_IF;
	      END_REGION FB_VALIDATE_INPUT

	    #FB_STATE_TCP_CONNECTING: //Wait for TCP to be established
	      REGION FB_TCP_CONNECTING
	        //Check process:
	        IF #tempTsendcError = TRUE THEN //when error:
	          #statTsendcEnable := FALSE; //disable TsendC
	          #statEnableTimerCommandWatchdog := FALSE;
	          #statStatus := #ERR_TCON_FAILED; // Set correct status that identifies error clearly
	          #statSubfunctionStatus := #tempTsendcStatus; // Status or return value of called FBs, FCs and system blocks
	          #statFBErrorState := #statFBState; // Set error state number for diagnostic
	          #statErrorUserCleared := TRUE;
	        ELSIF #tempTsendcStatus = #TSENDC_EST_OK THEN //when successfull:
	          //     Communication connection established.
	          #statEnableTimerCommandWatchdog := FALSE;
	          //Monitor Connection
	          #statFBState := #FB_STATE_OPERATING_MONITOR_TCP;
	          // Begin MQTT Connection
	          #statMqttConnectState := #MQTT_CONNECT_STATE_BUILD_PAKET;
	          //set status
	          #statStatus := #STATUS_MQTT_CONNECTING;
	        ELSIF #instTimerCommandWatchdog.Q THEN
	          #statTsendcEnable := FALSE; //disable TsendC
	          #statEnableTimerCommandWatchdog := FALSE;
	          #statStatus := #ERR_TCON_TIMEOUT; // Set correct status that identifies error clearly
	          #statSubfunctionStatus := #ERR_TCON_TIMEOUT; // Status or return value of called FBs, FCs and system blocks
	          #statFBErrorState := #statFBState; // Set error state number for diagnostic
	          #statErrorUserCleared := TRUE;
	        END_IF;
	      END_REGION FB_TCP_CONNECTING
	    #FB_STATE_OPERATING_MONITOR_TCP: // Processing active
	      REGION FB_OPERATING_MONITOR_TCP
	        //Reset Status on Msg Output - will be set when a new message is completly processed and ready at outputs.
	        #statRcvMsgStatus := #MSG_DECODE_STATUS_NO_NEW_MSG;
	        //Reset TsendC Req from last  cycle Request:

	        #statTsendcReq := FALSE;

	        //Monitor Connection - if disconnect occured:
	        IF ((#tempTsendcStatus > #TSENDC_COM_CLOSED AND #tempTsendcStatus < #TSENDC_EST_OK) //Status connection interupt
	          OR #tempTsendcError = TRUE) // Or error
	          AND #tempTrcvNdr = FALSE // And no new data (to see if broker send information why connection was interrupted)
	        THEN
	          REGION CONNECTION_INTERRUPTED
	            //Status reconnecting
	            //SET MQTT to no operation
	            #statMqttConnectState := #MQTT_CONNECT_STATE_NO_PROCESSING;
	            #statMqttCommandState := #MQTT_COMMAND_STATE_NO_PROCESSING;
	            #statRcvMsgDecodeState := #MSG_DECODE_STATE_NO_PROCESSING;
	            //Reset Pub ack
	            #statSendPubAckMsg := FALSE;
	            //reset Done bit if still set, regardless of input:
	            #statDone := FALSE;
	            //reset Watchdog
	            #statEnableTimerCommandWatchdog := FALSE;
	            // reset headerEncode
	            #statPaketHeaderEncodeDone := FALSE;
	            //set error  information
	            #statStatus := #ERR_TCP_RECONNECTING; // Set correct status that identifies error clearly
	            #statSubfunctionStatus := #tempTsendcStatus;// Status or return value of called FBs, FCs and system blocks
	            #statFBErrorState := #statFBState; // Set error state number for diagnostic
	            #statErrorAutoCleared := TRUE;
	            //Wait for reconect - next state
	            #statFBState := #FB_STATE_TCP_RECONNECTING;
	          END_REGION REGION CONNECTION_INTERRUPTED
	        ELSE
	          //Connection is OK
	          //Sending and receiving works
	          //Check Trcv Buffer for new Data
	          IF #tempTrcvNdr THEN
	            REGION TRCV_NEW_DATA
	              //Evaluate the TrcvBuffer, reset buffer pos to start
	              #tempTrcvBufferPos := 0;
	              // Parse the whole RCV Buffer
	              WHILE #tempTrcvBufferPos < (UDINT_TO_DINT(#tempTrcvRcvdLen)) DO
	                // Parse the whole RCV Buffer, check wether header or decoding
	                IF #statRcvMsgDecodeState = #MSG_DECODE_STATE_NO_PROCESSING THEN
	                  //If no decoding is in progress, look for new message header
	                  #tempRcvMsgTypeCase := #statRcvBuffer[#tempTrcvBufferPos] AND #BIT_MASK_HIGHBITS;
	                ELSE
	                  //decode is in progress, go directly to decoding
	                  #tempRcvMsgTypeCase := #MQTT_MSG_DECODING;
	                END_IF;

	                CASE #tempRcvMsgTypeCase OF
	                  #MQTT_MSG_TYPE_CONNACK:  // Statement section case 1
	                    REGION RECEIVED_CONACK_PACKET
	                      #tempTrcvBufferPos += 1;
	                      IF #statRcvBuffer[#tempTrcvBufferPos] = #REMAINING_LEN_2 //remainng Length must be 2;
	                      THEN //
	                        #tempTrcvBufferPos += 1;
	                        //byte one is 0000 000X where X is if Session was set // so depending on clean session or not  evaluate answer of server
	                        IF #statRcvBuffer[#tempTrcvBufferPos] = #MQTT_NO_SESSION_PRESENT THEN
	                          #tempTrcvBufferPos += 1;
	                          //VALID Answer, check code
	                          IF #statRcvBuffer[#tempTrcvBufferPos] = #MQTT_CONNACK_ACCEPTED
	                          THEN
	                            //All good
	                            #tempTrcvBufferPos += 1;
	                            #tempMqttConnAckRcvStatus := #RESPONSE_GOOD; //evaluate in MQTT StateMachine Below the response
	                          ELSE
	                            //NOT VALID CONNACK from server shows session has a bad return code
	                            #statStatus := #ERR_MQTT_CONNACK_RETURN_CODE_INVALID; // Set correct status that identifies error clearly
	                            #statSubfunctionStatus := #statRcvBuffer[#tempTrcvBufferPos]; // Status or return value of called FBs, FCs and system blocks
	                            #statFBErrorState := #statFBState; // Set error state number for diagnostic
	                            #statErrorUserCleared := TRUE;
	                            // Exit loop
	                            EXIT;
	                          END_IF;
	                        ELSE
	                          //NOT VALID, CONNACK from server shows session present
	                          #statStatus := #ERR_MQTT_CONNACK_INVALID_SESSION_FLAG; // Set correct status that identifies error clearly
	                          #statSubfunctionStatus := #ERR_MQTT_CONNACK_INVALID_SESSION_FLAG; // Status or return value of called FBs, FCs and system blocks
	                          #statFBErrorState := #statFBState; // Set error state number for diagnostic
	                          #statErrorUserCleared := TRUE;
	                          // Exit loop
	                          EXIT;
	                        END_IF;
	                      ELSE // We got a CONNACK paket, but remaining length was not 2 (Error)
	                        #statStatus := #ERR_MQTT_REM_LEN_INVALID; // Set correct status that identifies error clearly
	                        #statSubfunctionStatus := #ERR_MQTT_REM_LEN_INVALID; // Status or return value of called FBs, FCs and system blocks
	                        #statFBErrorState := #statFBState; // Set error state number for diagnostic
	                        #statErrorUserCleared := TRUE;
	                        // Exit loop
	                        EXIT;
	                      END_IF;
	                    END_REGION RECEIVED_CONACK_PACKET

	                  #MQTT_MSG_TYPE_PINGRESP:
	                    REGION RECEIVED_PINGRESP_PACKET
	                      #tempTrcvBufferPos += 1;
	                      IF #statRcvBuffer[#tempTrcvBufferPos] = #REMAINIG_LEN_0 //remainng Length must be 0;
	                      THEN
	                        #tempTrcvBufferPos += 1;
	                        #tempMqttPingRspRcv := #RESPONSE_GOOD; //evaluate in MQTT StateMachine Below the response
	                      ELSE// We got a Pingrsp paket, but remaining length was not 0 (Error)
	                        #statStatus := #ERR_MQTT_REM_LEN_INVALID; // Set correct status that identifies error clearly
	                        #statSubfunctionStatus := #ERR_MQTT_REM_LEN_INVALID; // Status or return value of called FBs, FCs and system blocks
	                        #statFBErrorState := #statFBState; // Set error state number for diagnostic
	                        #statErrorUserCleared := TRUE;
	                        // Exit loop
	                        EXIT;
	                      END_IF;
	                    END_REGION RECEIVED_PINGRESP_PAKET

	                  #MQTT_MSG_TYPE_PUBACK:
	                    REGION RECEIVED_PUBACK_PAKET
	                      #tempTrcvBufferPos += 1;
	                      IF #statRcvBuffer[#tempTrcvBufferPos] = #REMAINING_LEN_2 //remainng Length must be 2;
	                      THEN //
	                        #tempTrcvBufferPos += 1;
	                        #tempWordForSliceAddress := UINT_TO_WORD(#statPaketId);
	                        IF #statRcvBuffer[#tempTrcvBufferPos] = #tempWordForSliceAddress.%B1 THEN
	                          #tempTrcvBufferPos += 1;
	                          IF #statRcvBuffer[#tempTrcvBufferPos] = #tempWordForSliceAddress.%B0 THEN
	                            #tempTrcvBufferPos += 1;
	                            #tempMqttPubAckRcv := #RESPONSE_GOOD;
	                          ELSE
	                            #tempTrcvBufferPos += 1;
	                            #tempMqttPubAckRcv := #RESPONSE_PAKET_ID_INVALID;
	                          END_IF;
	                        ELSE
	                          #tempTrcvBufferPos += 1;
	                          #tempMqttPubAckRcv := #RESPONSE_PAKET_ID_INVALID;
	                        END_IF;
	                      ELSE
	                        #statStatus := #ERR_MQTT_REM_LEN_INVALID; // Set correct status that identifies error clearly
	                        #statSubfunctionStatus := #ERR_MQTT_REM_LEN_INVALID; // Status or return value of called FBs, FCs and system blocks
	                        #statFBErrorState := #statFBState; // Set error state number for diagnostic
	                        #statErrorUserCleared := TRUE;
	                        // Exit loop
	                        EXIT;
	                      END_IF;
	                    END_REGION RECEIVED_PUBACK_PAKET

	                  #MQTT_MSG_TYPE_PUBREC:
	                    REGION RECEIVED_PUBREC_PAKET
	                      #tempTrcvBufferPos += 1;
	                      IF #statRcvBuffer[#tempTrcvBufferPos] = #REMAINING_LEN_2 //remainng Length must be 2;
	                      THEN //
	                        #tempTrcvBufferPos += 1;
	                        #tempWordForSliceAddress := UINT_TO_WORD(#statPaketId);
	                        IF #statRcvBuffer[#tempTrcvBufferPos] = #tempWordForSliceAddress.%B1 THEN
	                          #tempTrcvBufferPos += 1;
	                          IF #statRcvBuffer[#tempTrcvBufferPos] = #tempWordForSliceAddress.%B0 THEN
	                            #tempTrcvBufferPos += 1;
	                            #statMqttPubRecRcv := #RESPONSE_GOOD;
	                          ELSE
	                            #tempTrcvBufferPos += 1;
	                            #statMqttPubRecRcv := #RESPONSE_PAKET_ID_INVALID;
	                          END_IF;
	                        ELSE
	                          #tempTrcvBufferPos += 1;
	                          #statMqttPubRecRcv := #RESPONSE_PAKET_ID_INVALID;
	                        END_IF;
	                      ELSE
	                        #statStatus := #ERR_MQTT_REM_LEN_INVALID; // Set correct status that identifies error clearly
	                        #statSubfunctionStatus := #ERR_MQTT_REM_LEN_INVALID; // Status or return value of called FBs, FCs and system blocks
	                        #statFBErrorState := #statFBState; // Set error state number for diagnostic
	                        #statErrorUserCleared := TRUE;
	                        // Exit loop
	                        EXIT;
	                      END_IF;
	                    END_REGION RECEIVED_PUBREC_PAKET

	                  #MQTT_MSG_TYPE_PUBCOMP:
	                    REGION RECEIVED_PUBCOMP_PAKET
	                      #tempTrcvBufferPos += 1;
	                      IF #statRcvBuffer[#tempTrcvBufferPos] = #REMAINING_LEN_2 //remainng Length must be 2;
	                      THEN //
	                        #tempTrcvBufferPos += 1;
	                        #tempWordForSliceAddress := UINT_TO_WORD(#statPaketId);
	                        IF #statRcvBuffer[#tempTrcvBufferPos] = #tempWordForSliceAddress.%B1 THEN
	                          #tempTrcvBufferPos += 1;
	                          IF #statRcvBuffer[#tempTrcvBufferPos] = #tempWordForSliceAddress.%B0 THEN
	                            #tempTrcvBufferPos += 1;
	                            #tempMqttPubCompRcv := #RESPONSE_GOOD;

	                          ELSE
	                            #tempTrcvBufferPos += 1;
	                            #tempMqttPubCompRcv := #RESPONSE_PAKET_ID_INVALID;

	                          END_IF;
	                        ELSE
	                          #tempTrcvBufferPos += 1;
	                          #tempMqttPubCompRcv := #RESPONSE_PAKET_ID_INVALID;

	                        END_IF;
	                      ELSE
	                        #statStatus := #ERR_MQTT_REM_LEN_INVALID; // Set correct status that identifies error clearly
	                        #statSubfunctionStatus := #ERR_MQTT_REM_LEN_INVALID; // Status or return value of called FBs, FCs and system blocks
	                        #statFBErrorState := #statFBState; // Set error state number for diagnostic
	                        #statErrorUserCleared := TRUE;
	                        // Exit loop
	                        EXIT;
	                      END_IF;
	                    END_REGION RECEIVED_PUBCOMP_PAKET

	                  #MQTT_MSG_TYPE_SUBACK:
	                    REGION RECEIVED_SUBACK_PAKET
	                      #tempTrcvBufferPos += 1;
	                      IF #statRcvBuffer[#tempTrcvBufferPos] = #REMAINING_LEN_3 //remainng Length must be 3;
	                      THEN //
	                        #tempTrcvBufferPos += 1;
	                        #tempWordForSliceAddress := UINT_TO_WORD(#statPaketId);
	                        IF #statRcvBuffer[#tempTrcvBufferPos] = #tempWordForSliceAddress.%B1 THEN
	                          #tempTrcvBufferPos += 1;
	                          IF #statRcvBuffer[#tempTrcvBufferPos] = #tempWordForSliceAddress.%B0 THEN
	                            #tempTrcvBufferPos += 1;
	                            IF #statRcvBuffer[#tempTrcvBufferPos] = #SUBSCRIBE_FAILURE THEN
	                              #tempTrcvBufferPos += 1;
	                              #tempMqttSubAckRcv := #RESPONSE_SUBSCRIBE_FAILED;
	                            ELSE
	                              #tempTrcvBufferPos += 1;
	                              #tempMqttSubAckRcv := #RESPONSE_GOOD;
	                            END_IF;
	                          ELSE
	                            #tempTrcvBufferPos += 1;
	                            #tempMqttSubAckRcv := #RESPONSE_PAKET_ID_INVALID;
	                          END_IF;
	                        ELSE
	                          #tempTrcvBufferPos += 1;
	                          #tempMqttSubAckRcv := #RESPONSE_PAKET_ID_INVALID;
	                        END_IF;
	                      ELSE
	                        #statStatus := #ERR_MQTT_REM_LEN_INVALID; // Set correct status that identifies error clearly
	                        #statSubfunctionStatus := #ERR_MQTT_REM_LEN_INVALID; // Status or return value of called FBs, FCs and system blocks
	                        #statFBErrorState := #statFBState; // Set error state number for diagnostic
	                        #statErrorUserCleared := TRUE;
	                        // Exit loop
	                        EXIT;
	                      END_IF;
	                    END_REGION RECEIVED_SUBACK_PAKET

	                  #MQTT_MSG_TYPE_UNSUBACK:
	                    REGION RECEIVED_UNSUBACK_PAKET
	                      #tempTrcvBufferPos += 1;
	                      IF #statRcvBuffer[#tempTrcvBufferPos] = #REMAINING_LEN_2 //remainng Length must be 2;
	                      THEN //
	                        #tempTrcvBufferPos += 1;
	                        #tempWordForSliceAddress := UINT_TO_WORD(#statPaketId);
	                        IF #statRcvBuffer[#tempTrcvBufferPos] = #tempWordForSliceAddress.%B1 THEN
	                          #tempTrcvBufferPos += 1;
	                          IF #statRcvBuffer[#tempTrcvBufferPos] = #tempWordForSliceAddress.%B0 THEN
	                            #tempTrcvBufferPos += 1;
	                            #tempMqttUnSubAckRcv := #RESPONSE_GOOD;
	                          ELSE
	                            #tempTrcvBufferPos += 1;
	                            #tempMqttUnSubAckRcv := #RESPONSE_PAKET_ID_INVALID;
	                          END_IF;
	                        ELSE
	                          #tempTrcvBufferPos += 1;
	                          #tempMqttUnSubAckRcv := #RESPONSE_PAKET_ID_INVALID;
	                        END_IF;
	                      ELSE
	                        #statStatus := #ERR_MQTT_REM_LEN_INVALID; // Set correct status that identifies error clearly
	                        #statSubfunctionStatus := #ERR_MQTT_REM_LEN_INVALID; // Status or return value of called FBs, FCs and system blocks
	                        #statFBErrorState := #statFBState; // Set error state number for diagnostic
	                        #statErrorUserCleared := TRUE;
	                        // Exit loop
	                        EXIT;
	                      END_IF;
	                    END_REGION RECEIVED_UNSUBACK_PAKET

	                  #MQTT_MSG_TYPE_RCV_PUB_MESSAGE:
	                    REGION RECEIVED_PUBLISH_PAKET_FROM_BROKER
	                      //Received a message, start process.
	                      //init
	                      #tempMultiplierToDecode := #INIT_UDINT_1;
	                      #statRcvMsgInternalStatus := #MSG_DECODE_STATUS_NO_NEW_MSG;
	                      #statRcvMsgTotalLen := 0;
	                      #statRcvMsgTopicLen := 0;
	                      #statRcvMsgPayloadLen := 0;
	                      //Check and store QoS for later use
	                      IF (#statRcvBuffer[#tempTrcvBufferPos] AND #BIT_MASK_QOS) = #MQTT_MSG_TYPE_RCV_PUB_MESSAGE_QoS0
	                      THEN
	                        #statRcvMsgQoS := #MQTT_QOS_0;
	                      ELSIF (#statRcvBuffer[#tempTrcvBufferPos] AND #BIT_MASK_QOS) = #MQTT_MSG_TYPE_RCV_PUB_MESSAGE_QoS1
	                      THEN
	                        #statRcvMsgQoS := #MQTT_QOS_1;
	                      ELSIF (#statRcvBuffer[#tempTrcvBufferPos] AND #BIT_MASK_QOS) = #MQTT_MSG_TYPE_RCV_PUB_MESSAGE_QoS2
	                      THEN
	                        #statRcvMsgQoS := #MQTT_QOS_2;
	                      ELSIF (#statRcvBuffer[#tempTrcvBufferPos] AND #BIT_MASK_QOS) = #MQTT_MSG_TYPE_RCV_PUB_MESSAGE_BAD
	                      THEN
	                        #statStatus := #ERR_MQTT_MALFORMED_QOS_RECEIVED; // Set correct status that identifies error clearly
	                        #statSubfunctionStatus := #ERR_MQTT_MALFORMED_QOS_RECEIVED; // Status or return value of called FBs, FCs and system blocks
	                        #statFBErrorState := #statFBState; // Set error state number for diagnostic
	                        #statErrorUserCleared := TRUE;
	                        // Exit loop
	                        EXIT;
	                      END_IF;

	                      //Calculate total publish len (topic,paketid,payload)
	                      REPEAT
	                        #tempTrcvBufferPos += 1; //Increment
	                        #statRcvMsgTotalLen += BYTE_TO_UDINT((#statRcvBuffer[#tempTrcvBufferPos] AND #DEFAULT_MULTIPLIER_BYTE_127)) * #tempMultiplierToDecode;
	                        #tempMultiplierToDecode *= #SEND_LEN_MULTIPLIER_UDINT_128;
	                        IF (#tempMultiplierToDecode > #MAX_ALLOWED_PAKET_SIZE)
	                        THEN//Throw error here // Malformed remain length.
	                          #statStatus := #ERR_MQTT_REM_LEN_INVALID; // Set correct status that identifies error clearly
	                          #statSubfunctionStatus := #ERR_MQTT_REM_LEN_INVALID; // Status or return value of called FBs, FCs and system blocks
	                          #statFBErrorState := #statFBState; // Set error state number for diagnostic
	                          #statErrorUserCleared := TRUE;
	                          // Exit loop
	                          EXIT;
	                        END_IF;
	                      UNTIL ((#statRcvBuffer[#tempTrcvBufferPos] AND UDINT_TO_BYTE(#SEND_LEN_MULTIPLIER_UDINT_128)) = 0)
	                      END_REPEAT;
	                      #tempTrcvBufferPos += 1; //Increment
	                      //#statIncPaketRemLen contains total paket len
	                      //Save Topic Len
	                      #tempWordForSliceAddress.%B1 := #statRcvBuffer[#tempTrcvBufferPos]; //MSB
	                      #tempTrcvBufferPos += 1; //Increment
	                      #tempWordForSliceAddress.%B0 := #statRcvBuffer[#tempTrcvBufferPos]; //LSB
	                      #tempTrcvBufferPos += 1; //Increment
	                      #statRcvMsgTopicLen := WORD_TO_UINT(#tempWordForSliceAddress);
	                      //Set Payload len
	                      IF #statRcvMsgQoS = #MQTT_QOS_0 THEN
	                        //Payload Len is total Len minus topic len minus topic len info
	                        #statRcvMsgPayloadLen := #statRcvMsgTotalLen - #statRcvMsgTopicLen - #TWO_BYTE_LEN_INFO;
	                      ELSE
	                        //PayloadLen is total Len minus topic len minus topic len info minus paket Id len
	                        #statRcvMsgPayloadLen := #statRcvMsgTotalLen - #statRcvMsgTopicLen - #TWO_BYTE_LEN_INFO - #TWO_BYTE_LEN_INFO;
	                      END_IF;

	                      //Clear Output message:
	                      #receivedTopic := #EMPTY_WSTRING;
	                      //Start receiving with topic
	                      #statRcvMsgDecodeState := #MSG_DECODE_STATE_TOPIC;
	                      //Start Topic at first character
	                      #statRcvMsgTopicPos := #FIRST_CHARACTER;
	                      //Start RcvMsg at first array element
	                      #statRcvMsgPayloadPos := LOWER_BOUND(ARR := #receivedMsgPayload, DIM := #ONE_DIMENSION);
	                      //Set Output for received len according to array dimension
	                      #tempReceivedMsgDataArrayTotalLen := ABS(UPPER_BOUND(ARR := #receivedMsgPayload, DIM := #ONE_DIMENSION) - LOWER_BOUND(ARR := #receivedMsgPayload, DIM := #ONE_DIMENSION)) + #ARRAY_LEN_OFFSET_PLUS_1;
	                      IF #statRcvMsgPayloadLen < #tempReceivedMsgDataArrayTotalLen THEN
	                        #statRcvMsgDataLen := #statRcvMsgPayloadLen;
	                      ELSE
	                        #statRcvMsgDataLen := DINT_TO_UDINT(#tempReceivedMsgDataArrayTotalLen);
	                      END_IF;
	                    END_REGION RECEIVED_PUBLISH_PAKET_FROM_BROKER

	                  #MQTT_MSG_DECODING:
	                    REGION RECEIVED_PAKET_DECODE
	                      CASE #statRcvMsgDecodeState OF
	                        #MSG_DECODE_STATE_NO_PROCESSING: // NO Processing
	                          ;
	                        #MSG_DECODE_STATE_TOPIC:  // Statement section case 1
	                          #tempReceivedTopicStringMaxLen := MAX_LEN(#receivedTopic);
	                          //Copy Topic To WString Inout
	                          IF #statRcvMsgTopicPos <= #tempReceivedTopicStringMaxLen THEN
	                            #receivedTopic[#statRcvMsgTopicPos] := BYTE_TO_WCHAR(#statRcvBuffer[#tempTrcvBufferPos]);
	                            #statRcvMsgTopicPos += 1;
	                          ELSE
	                            //Max String len reached.
	                            #statRcvMsgInternalStatus := #MSG_DECODE_STATUS_TOPIC_TOO_LONG;
	                          END_IF;
	                          //decrement
	                          #statRcvMsgTopicLen -= 1;
	                          //increment
	                          #tempTrcvBufferPos += 1;
	                          //Check condition, if topic fully decoded:
	                          IF #statRcvMsgTopicLen <= 0 THEN
	                            //Decide what to do next:
	                            IF #statRcvMsgQoS > #MQTT_QOS_0 THEN
	                              //NextStep Decode PaketID
	                              #statRcvMsgDecodeState := #MSG_DECODE_STATE_PAKET_ID_MSB;
	                            ELSIF #statRcvMsgQoS = #MQTT_QOS_0 AND #statRcvMsgPayloadLen > 0 THEN
	                              //NextStep Decode Payload
	                              #statRcvMsgDecodeState := #MSG_DECODE_STATE_PAYLOAD;
	                            ELSE
	                              // QoS=0 and no Payload => Done
	                              // Decoding complete
	                              #statRcvMsgDecodeState := #MSG_DECODE_STATE_NO_PROCESSING;
	                              //Set New message flag
	                              IF #statRcvMsgInternalStatus = #MSG_DECODE_STATUS_NO_NEW_MSG THEN
	                                //New message received ok
	                                #statRcvMsgStatus := #MSG_DECODE_STATUS_NEW_MSG_OK;
	                              ELSE
	                                //Message received, but Payload or Topic longer than inout data area
	                                #statRcvMsgStatus := #MSG_DECODE_STATUS_TOPIC_TOO_LONG;
	                              END_IF;
	                            END_IF;
	                          END_IF;
	                        #MSG_DECODE_STATE_PAKET_ID_MSB:  // Decode PaketId MSB
	                          //Copy PaketID
	                          #statRcvMsgPaketId.%B1 := #statRcvBuffer[#tempTrcvBufferPos]; //MSB
	                          #tempTrcvBufferPos += 1; //Increment
	                          #statRcvMsgDecodeState := #MSG_DECODE_STATE_PAKET_ID_LSB;
	                        #MSG_DECODE_STATE_PAKET_ID_LSB: // Decode PaketId LSB
	                          //Copy PaketID
	                          #statRcvMsgPaketId.%B0 := #statRcvBuffer[#tempTrcvBufferPos]; //LSB
	                          #tempTrcvBufferPos += 1; //Increment
	                          IF #statRcvMsgPayloadLen > 0 THEN
	                            #statRcvMsgDecodeState := #MSG_DECODE_STATE_PAYLOAD;
	                          ELSE
	                            // Decoding complete
	                            #statRcvMsgDecodeState := #MSG_DECODE_STATE_NO_PROCESSING;
	                            //Set New message flag
	                            IF #statRcvMsgInternalStatus = #MSG_DECODE_STATUS_NO_NEW_MSG THEN
	                              //New message received ok
	                              #statRcvMsgStatus := #MSG_DECODE_STATUS_NEW_MSG_OK;
	                            ELSE
	                              //Message received, but Payload or Topic longer than inout data area
	                              #statRcvMsgStatus := #MSG_DECODE_STATUS_TOPIC_TOO_LONG;
	                            END_IF;
	                            // Send PubAck Msg
	                            #statSendPubAckMsg := TRUE;
	                          END_IF;
	                        #MSG_DECODE_STATE_PAYLOAD:
	                          #tempUpperBoundRcvMsgDataArray := UPPER_BOUND(ARR := #receivedMsgPayload, DIM := #ONE_DIMENSION);

	                          IF #statRcvMsgPayloadPos <= #tempUpperBoundRcvMsgDataArray THEN
	                            //Copy to output
	                            #receivedMsgPayload[#statRcvMsgPayloadPos] := (#statRcvBuffer[#tempTrcvBufferPos]);
	                            //Increment the pos
	                            #statRcvMsgPayloadPos += 1;
	                          ELSE
	                            //Max Payload len reached, skip
	                            #statRcvMsgInternalStatus := #MSG_DECODE_STATUS_PAYLOAD_TOO_LONG;
	                          END_IF;
	                          //Decrement msg payload len
	                          #statRcvMsgPayloadLen -= 1;
	                          //Increment Buffer Pos
	                          #tempTrcvBufferPos += 1;
	                          //Check condition, if payload fully decoded:
	                          IF #statRcvMsgPayloadLen <= 0 THEN
	                            // Decoding complete
	                            #statRcvMsgDecodeState := #MSG_DECODE_STATE_NO_PROCESSING;
	                            //Set New message flag
	                            IF #statRcvMsgInternalStatus = #MSG_DECODE_STATUS_NO_NEW_MSG THEN
	                              //New message received ok
	                              #statRcvMsgStatus := #MSG_DECODE_STATUS_NEW_MSG_OK;
	                            ELSE
	                              //Message received, but Payload or Topic longer than inout data area
	                              #statRcvMsgStatus := #MSG_DECODE_STATUS_PAYLOAD_TOO_LONG;
	                            END_IF;
	                            //Decide if a PUB ACK needs to be send
	                            IF #statRcvMsgQoS > #MQTT_QOS_0 THEN
	                              // Send PubAck Msg
	                              #statSendPubAckMsg := TRUE;
	                            END_IF;
	                          END_IF;
	                        ELSE
	                          //else case
	                          #statStatus := #ERR_UNDEFINED_STATE;
	                          #statErrorUserCleared := TRUE;
	                          ;
	                      END_CASE;
	                    END_REGION RECEIVED_PAKET_DECODE
	                  ELSE // No Header found, SKIP entry of buffer:
	                    #tempTrcvBufferPos += 1;
	                END_CASE;
	              END_WHILE;
	            END_REGION TRCV_NEW_DATA
	          END_IF;

	          //Send an Publish Acknowledge Msg, if necessary
	          REGION SEND_PUB_ACK_MSG_ON_SUBSCRIPTIONS
	            //Send Acknowledgements to Subscribed messages, if requested (QoS =1)
	            IF #statSendPubAckMsg = TRUE AND // send pub ack Request
	              #statMqttCommandState = #MQTT_COMMAND_STATE_NO_PROCESSING AND // no send job processing
	              #tempTsendcBusy = FALSE AND // tsendC is ready
	              #tempTsendcDone = FALSE // tsendC did not finished in this cycle
	            THEN
	              //Set Pos
	              #statSendBufferPos := 0;
	              //Write Msg Type
	              #statSendBuffer[#statSendBufferPos] := #MQTT_MSG_TYPE_PUBACK;
	              #statSendBufferPos += 1;
	              //Write Msg Len
	              #statSendBuffer[#statSendBufferPos] := #REMAINING_LEN_2;
	              #statSendBufferPos += 1;
	              //Write Paket Id - first MSB then LSB
	              #statSendBuffer[#statSendBufferPos] := #statRcvMsgPaketId.%B1;
	              #statSendBufferPos += 1;
	              #statSendBuffer[#statSendBufferPos] := #statRcvMsgPaketId.%B0;
	              #statSendBufferPos += 1;
	              //Set Send Len:
	              #statTsendcLen := #statSendBufferPos;
	              //Send msg
	              #statTsendcReq := TRUE;
	              //Reset ack:
	              #statSendPubAckMsg := FALSE;
	            END_IF;
	          END_REGION SEND_PUB_ACK_MSG_ON_SUBSCRIPTIONS

	          REGION MQTT_STATE_MACHINE
	            CASE #statMqttConnectState OF
	              #MQTT_CONNECT_STATE_NO_PROCESSING:  // Statement section case 1
	                ;
	              #MQTT_CONNECT_STATE_BUILD_PAKET:  //
	                REGION BUILD_CONNECT_PAKET
	                  //Remaining Length is the length of the variable header (10 bytes) plus the length of the Payload.
	                  //Max Len of Mqtt pakets is per Standard 268,435,455 Bytes (ff,ff,ff,7f)
	                  //Calculate Remain Len will be 10 bytes
	                  //plus Len of ClientId   (max 3*16382 WChars= 49.146 Bytes)
	                  //plus Len of User (max 3*16382 WChars= 49.146 Bytes)
	                  //plus Len of PW (max 3*16382 WChars= 49.146 Bytes)
	                  //plus Len of WillTopic (max 3*16382 WChars= 49.146 Bytes)
	                  //plus Len of WillMessage (max 65535 Bytes - as only 2 Bytes Len info is possible)
	                  // = Total 262 119 Bytes


	                  // Must obey, if not currently sending PubAck Msg on a subscription
	                  // Else, try in the next cycle
	                  IF #tempTsendcBusy = FALSE AND // tsendC is ready
	                    #tempTsendcDone = FALSE AND  // tsendC did not finish in this cycle
	                    #statTsendcReq = FALSE THEN // no request from pub ack request

	                    //Only need to encode header once
	                    IF #statPaketHeaderEncodeDone = FALSE THEN
	                      // INIT
	                      #statSendBufferPos := 0;
	                      #statClientIdPos := #FIRST_CHARACTER;
	                      #statClientIdEncodeState := #FIRST_ENCODING;

	                      #statWillTopicEncodeState := #FIRST_ENCODING;
	                      #statWillTopicPos := #FIRST_CHARACTER;

	                      #statWillMessageEncodeState := #FIRST_ENCODING;
	                      #statWillMessagePos := 0; // The Posistion for the WILL Message Array

	                      #statUserNameEncodeState := #FIRST_ENCODING;
	                      #statUserNamePos := #FIRST_CHARACTER;

	                      #statPasswordEncodeState := #FIRST_ENCODING;
	                      #statPasswordPos := #FIRST_CHARACTER;

	                      #statSendPaketTotalRemLen := #CONNECT_HEADER_10BYTE_LEN;
	                      #statClientIdLenUtf8Encoded := 0;
	                      #statWillTopicLenUtf8Encoded := 0;
	                      #statUsernameLenUtf8Encoded := 0;
	                      #statPasswordLenUtf8Encoded := 0;
	                      //End Init

	                      // Encode Client ID Len
	                      // Client ID must always be present
	                      FOR #tempLoopCounter := #FIRST_CHARACTER TO LEN(#clientIdentifier) DO
	                        "LMQTT_ConvertToUtf8"(character     := #clientIdentifier[#tempLoopCounter],
	                                              convertedUtf8 => #tempConvertedUtf8,
	                                              bytesUsed     => #tempBytesUsedUtf8,
	                                              error         => #tempErrorConvertUtf8,
	                                              status        => #tempStatusConvertUtf8);
	                        #statClientIdLenUtf8Encoded := #statClientIdLenUtf8Encoded + #tempBytesUsedUtf8;
	                      END_FOR;

	                      #statSendPaketTotalRemLen := #statSendPaketTotalRemLen + #statClientIdLenUtf8Encoded + #TWO_BYTE_LEN_INFO;


	                      IF #username <> #EMPTY_WSTRING
	                      THEN
	                        #tempUserFlag := TRUE;
	                        FOR #tempLoopCounter := #FIRST_CHARACTER TO LEN(#username) DO
	                          "LMQTT_ConvertToUtf8"(character     := #username[#tempLoopCounter],
	                                                convertedUtf8 => #tempConvertedUtf8,
	                                                bytesUsed     => #tempBytesUsedUtf8,
	                                                error         => #tempErrorConvertUtf8,
	                                                status        => #tempStatusConvertUtf8);
	                          #statUsernameLenUtf8Encoded := #statUsernameLenUtf8Encoded + #tempBytesUsedUtf8;
	                        END_FOR;
	                        #statSendPaketTotalRemLen := #statSendPaketTotalRemLen + #statUsernameLenUtf8Encoded + #TWO_BYTE_LEN_INFO;
	                      ELSE
	                        #statUserNameEncodeState := #NOT_USED_NO_ENCODING;
	                        #tempUserFlag := FALSE;
	                      END_IF;

	                      IF #password <> #EMPTY_WSTRING AND #username <> #EMPTY_WSTRING
	                      THEN
	                        #tempPasswordFlag := TRUE;
	                        FOR #tempLoopCounter := #FIRST_CHARACTER TO LEN(#password) DO
	                          "LMQTT_ConvertToUtf8"(character     := #password[#tempLoopCounter],
	                                                convertedUtf8 => #tempConvertedUtf8,
	                                                bytesUsed     => #tempBytesUsedUtf8,
	                                                error         => #tempErrorConvertUtf8,
	                                                status        => #tempStatusConvertUtf8);
	                          #statPasswordLenUtf8Encoded := #statPasswordLenUtf8Encoded + #tempBytesUsedUtf8;
	                        END_FOR;
	                        #statSendPaketTotalRemLen := #statSendPaketTotalRemLen + #statPasswordLenUtf8Encoded + #TWO_BYTE_LEN_INFO;
	                      ELSE
	                        #statPasswordEncodeState := #NOT_USED_NO_ENCODING;
	                        #tempPasswordFlag := FALSE;
	                      END_IF;


	                      IF #willtopic <> #EMPTY_WSTRING
	                      THEN
	                        #tempWillFlag := TRUE;
	                        CASE #statWillQos OF
	                          #MQTT_QOS_0:  // Statement section case 1
	                            #tempWillQoS1 := FALSE;
	                            #tempWillQoS2 := FALSE;
	                          #MQTT_QOS_1:  // Statement section case 2 to 4
	                            #tempWillQoS1 := TRUE;
	                            #tempWillQoS2 := FALSE;
	                          #MQTT_QOS_2:
	                            #tempWillQoS1 := FALSE;
	                            #tempWillQoS2 := True;
	                          ELSE  // Statement section ELSE
	                            ;
	                        END_CASE;
	                        FOR #tempLoopCounter := #FIRST_CHARACTER TO LEN(#willtopic) DO
	                          // Statement section FOR
	                          "LMQTT_ConvertToUtf8"(character     := #willtopic[#tempLoopCounter],
	                                                convertedUtf8 => #tempConvertedUtf8,
	                                                bytesUsed     => #tempBytesUsedUtf8,
	                                                error         => #tempErrorConvertUtf8,
	                                                status        => #tempStatusConvertUtf8);
	                          #statWillTopicLenUtf8Encoded := #statWillTopicLenUtf8Encoded + #tempBytesUsedUtf8;
	                        END_FOR;
	                        //Add WillTopic Len and Will Message Len (and len info twice)
	                        #statSendPaketTotalRemLen := #statSendPaketTotalRemLen + #statWillTopicLenUtf8Encoded + #statWillMessageCnt + (2 * #TWO_BYTE_LEN_INFO);
	                      ELSE
	                        #statWillTopicEncodeState := #NOT_USED_NO_ENCODING;
	                        #statWillMessageEncodeState := #NOT_USED_NO_ENCODING;
	                        #tempWillFlag := FALSE;
	                        #statWillRetain := FALSE;
	                        #tempWillQoS1 := FALSE;
	                        #tempWillQoS2 := FALSE;
	                      END_IF;

	                      //Build Connect Telegram
	                      //Fixed Header - Write Paket Type
	                      #statSendBuffer[#statSendBufferPos] := #MQTT_MSG_TYPE_CONNECT; // 1 Byte
	                      #statSendBufferPos += 1; // increment

	                      //Write Remaining Paket Len info
	                      WHILE (#statSendPaketTotalRemLen > #DEFAULT_VALUE_ZERO)
	                      DO//See MQTT Spec for explanation of this calculation
	                        #statEncodedRemPaketLenAsByte := UDINT_TO_BYTE(#statSendPaketTotalRemLen MOD #SEND_LEN_MULTIPLIER_UDINT_128);
	                        #statSendPaketTotalRemLen := #statSendPaketTotalRemLen / #SEND_LEN_MULTIPLIER_UDINT_128;
	                        // if there are more data to encode, set the top bit of this byte
	                        IF #statSendPaketTotalRemLen > #DEFAULT_VALUE_ZERO
	                        THEN
	                          // Do this and continue while loop
	                          #statEncodedRemPaketLenAsByte := #statEncodedRemPaketLenAsByte OR UDINT_TO_BYTE(#SEND_LEN_MULTIPLIER_UDINT_128);
	                          #statSendBuffer[#statSendBufferPos] := #statEncodedRemPaketLenAsByte;
	                          #statSendBufferPos += 1;
	                        ELSE
	                          //do this and leave while loop
	                          #statSendBuffer[#statSendBufferPos] := #statEncodedRemPaketLenAsByte;
	                          #statSendBufferPos += 1;
	                        END_IF;
	                      END_WHILE;

	                      //Build Connect Telegram
	                      // Write Protocol name
	                      #statSendBuffer[#statSendBufferPos] := #CONN_PROTOCOL_NAME_0;
	                      #statSendBufferPos += 1;
	                      #statSendBuffer[#statSendBufferPos] := #CONN_PROTOCOL_NAME_4;
	                      #statSendBufferPos += 1;
	                      #statSendBuffer[#statSendBufferPos] := CHAR_TO_BYTE('M');
	                      #statSendBufferPos += 1;
	                      #statSendBuffer[#statSendBufferPos] := CHAR_TO_BYTE('Q');
	                      #statSendBufferPos += 1;
	                      #statSendBuffer[#statSendBufferPos] := CHAR_TO_BYTE('T');
	                      #statSendBufferPos += 1;
	                      #statSendBuffer[#statSendBufferPos] := CHAR_TO_BYTE('T');
	                      #statSendBufferPos += 1;
	                      //Write Protocol Level
	                      #statSendBuffer[#statSendBufferPos] := #CONN_PROTOCOL_MQTT_VERSION_3_1_1;
	                      #statSendBufferPos += 1;
	                      //Write Connect Flags
	                      #statSendBuffer[#statSendBufferPos].%X0 := false;
	                      #statSendBuffer[#statSendBufferPos].%X1 := True;
	                      #statSendBuffer[#statSendBufferPos].%X2 := #tempWillFlag;
	                      #statSendBuffer[#statSendBufferPos].%X3 := #tempWillQoS1;
	                      #statSendBuffer[#statSendBufferPos].%X4 := #tempWillQoS2;
	                      #statSendBuffer[#statSendBufferPos].%X5 := #statWillRetain;
	                      #statSendBuffer[#statSendBufferPos].%X6 := #tempPasswordFlag;
	                      #statSendBuffer[#statSendBufferPos].%X7 := #tempUserFlag;
	                      #statSendBufferPos += 1;
	                      //Write Keep Alive in sec
	                      #tempWordForSliceAddress := UINT_TO_WORD(#connParam.keepAlive);
	                      #statSendBuffer[#statSendBufferPos] := #tempWordForSliceAddress.%B1;
	                      #statSendBufferPos += 1;
	                      #statSendBuffer[#statSendBufferPos] := #tempWordForSliceAddress.%B0;
	                      #statSendBufferPos += 1;

	                      //Set To Complete this, can skip in further progess
	                      #statPaketHeaderEncodeDone := TRUE;
	                    END_IF;

	                    // Payload
	                    // These fields, if present, MUST appear in the order:
	                    // Client Identifier, Will topic, Will message, User Name, password


	                    //ClientIdentifier
	                    IF #statSendBufferPos <= #MAX_BUFFER_LEN_SEND - #TWO_BYTE_LEN_INFO THEN
	                      CASE #statClientIdEncodeState OF
	                        #FIRST_ENCODING:  // Statement section case 1
	                          //ADD len info into paket

	                          #tempWordForSliceAddress := UINT_TO_WORD(#statClientIdLenUtf8Encoded);
	                          #statSendBuffer[#statSendBufferPos] := #tempWordForSliceAddress.%B1; //MSB
	                          #statSendBufferPos += 1;
	                          #statSendBuffer[#statSendBufferPos] := #tempWordForSliceAddress.%B0; // LSB
	                          #statSendBufferPos += 1;

	                          FOR #tempLoopCounter := #statClientIdPos TO LEN(#clientIdentifier) DO
	                            "LMQTT_ConvertToUtf8"(character     := #clientIdentifier[#tempLoopCounter],
	                                                  convertedUtf8 => #tempConvertedUtf8,
	                                                  bytesUsed     => #tempBytesUsedUtf8,
	                                                  error         => #tempErrorConvertUtf8,
	                                                  status        => #tempStatusConvertUtf8);

	                            IF #statSendBufferPos + #tempBytesUsedUtf8 <= #MAX_BUFFER_LEN_SEND THEN
	                              #statClientIdPos += 1;
	                              CASE #tempBytesUsedUtf8 OF
	                                #UTF_1_BYTE_USED:  // Statement section case 1
	                                  #statSendBuffer[#statSendBufferPos] := #tempConvertedUtf8.%B0;
	                                  #statSendBufferPos += 1;
	                                #UTF_2_BYTE_USED:
	                                  #statSendBuffer[#statSendBufferPos] := #tempConvertedUtf8.%B0;
	                                  #statSendBufferPos += 1;
	                                  #statSendBuffer[#statSendBufferPos] := #tempConvertedUtf8.%B1;
	                                  #statSendBufferPos += 1;
	                                #UTF_3_BYTE_USED:  // Statement section case 2 to 4
	                                  #statSendBuffer[#statSendBufferPos] := #tempConvertedUtf8.%B0;
	                                  #statSendBufferPos += 1;
	                                  #statSendBuffer[#statSendBufferPos] := #tempConvertedUtf8.%B1;
	                                  #statSendBufferPos += 1;
	                                  #statSendBuffer[#statSendBufferPos] := #tempConvertedUtf8.%B2;
	                                  #statSendBufferPos += 1;
	                                ELSE  // Statement section ELSE
	                                  ;
	                              END_CASE;
	                            ELSE
	                              //When buffer full
	                              #statClientIdEncodeState := #SUBSEQUENT_ENCODING;
	                              EXIT;
	                            END_IF;
	                          END_FOR;
	                          IF #statClientIdPos >= LEN(#clientIdentifier) THEN
	                            #statClientIdEncodeState := #ENCODE_DONE;
	                          END_IF;


	                        #SUBSEQUENT_ENCODING:  // Statement section case 2 to 4
	                          FOR #tempLoopCounter := #statClientIdPos TO LEN(#clientIdentifier) DO
	                            "LMQTT_ConvertToUtf8"(character     := #clientIdentifier[#tempLoopCounter],
	                                                  convertedUtf8 => #tempConvertedUtf8,
	                                                  bytesUsed     => #tempBytesUsedUtf8,
	                                                  error         => #tempErrorConvertUtf8,
	                                                  status        => #tempStatusConvertUtf8);
	                            IF #statSendBufferPos + #tempBytesUsedUtf8 <= #MAX_BUFFER_LEN_SEND THEN
	                              #statClientIdPos += 1;
	                              CASE #tempBytesUsedUtf8 OF
	                                #UTF_1_BYTE_USED:  // Statement section case 1
	                                  #statSendBuffer[#statSendBufferPos] := #tempConvertedUtf8.%B0;
	                                  #statSendBufferPos += 1;
	                                #UTF_2_BYTE_USED:
	                                  #statSendBuffer[#statSendBufferPos] := #tempConvertedUtf8.%B0;
	                                  #statSendBufferPos += 1;
	                                  #statSendBuffer[#statSendBufferPos] := #tempConvertedUtf8.%B1;
	                                  #statSendBufferPos += 1;
	                                #UTF_3_BYTE_USED:  // Statement section case 2 to 4
	                                  #statSendBuffer[#statSendBufferPos] := #tempConvertedUtf8.%B0;
	                                  #statSendBufferPos += 1;
	                                  #statSendBuffer[#statSendBufferPos] := #tempConvertedUtf8.%B1;
	                                  #statSendBufferPos += 1;
	                                  #statSendBuffer[#statSendBufferPos] := #tempConvertedUtf8.%B2;
	                                  #statSendBufferPos += 1;
	                                ELSE  // Statement section ELSE
	                                  ;
	                              END_CASE;
	                            ELSE
	                              //When buffer full
	                              EXIT;
	                            END_IF;
	                          END_FOR;
	                          IF #statClientIdPos >= LEN(#clientIdentifier) THEN
	                            #statClientIdEncodeState := #ENCODE_DONE;
	                          END_IF;
	                        ELSE  // Statement section ELSE
	                          ; // IDLE / SKIP
	                      END_CASE;
	                    END_IF;

	                    // Will Topic
	                    // If the Will Flag is set to 1, the Will Topic is the next field in the payload. It must be > 0 Bytes

	                    IF #statClientIdEncodeState = #ENCODE_DONE
	                      AND #statSendBufferPos <= #MAX_BUFFER_LEN_SEND - #TWO_BYTE_LEN_INFO THEN
	                      //When Client Id is encoded and buffer not full
	                      //And willTopic is used
	                      CASE #statWillTopicEncodeState OF
	                        #FIRST_ENCODING:  // Statement section case 1
	                          //ADD len info into paket

	                          #tempWordForSliceAddress := UINT_TO_WORD(#statWillTopicLenUtf8Encoded);
	                          #statSendBuffer[#statSendBufferPos] := #tempWordForSliceAddress.%B1; //MSB
	                          #statSendBufferPos += 1;
	                          #statSendBuffer[#statSendBufferPos] := #tempWordForSliceAddress.%B0; // LSB
	                          #statSendBufferPos += 1;

	                          FOR #tempLoopCounter := #statWillTopicPos TO LEN(#willtopic) DO
	                            "LMQTT_ConvertToUtf8"(character     := #willtopic[#tempLoopCounter],
	                                                  convertedUtf8 => #tempConvertedUtf8,
	                                                  bytesUsed     => #tempBytesUsedUtf8,
	                                                  error         => #tempErrorConvertUtf8,
	                                                  status        => #tempStatusConvertUtf8);

	                            IF #statSendBufferPos + #tempBytesUsedUtf8 <= #MAX_BUFFER_LEN_SEND THEN
	                              //Increment when successful
	                              #statWillTopicPos += 1;

	                              CASE #tempBytesUsedUtf8 OF
	                                #UTF_1_BYTE_USED:  // Statement section case 1
	                                  #statSendBuffer[#statSendBufferPos] := #tempConvertedUtf8.%B0;
	                                  #statSendBufferPos += 1;
	                                #UTF_2_BYTE_USED:
	                                  #statSendBuffer[#statSendBufferPos] := #tempConvertedUtf8.%B0;
	                                  #statSendBufferPos += 1;
	                                  #statSendBuffer[#statSendBufferPos] := #tempConvertedUtf8.%B1;
	                                  #statSendBufferPos += 1;
	                                #UTF_3_BYTE_USED:  // Statement section case 2 to 4
	                                  #statSendBuffer[#statSendBufferPos] := #tempConvertedUtf8.%B0;
	                                  #statSendBufferPos += 1;
	                                  #statSendBuffer[#statSendBufferPos] := #tempConvertedUtf8.%B1;
	                                  #statSendBufferPos += 1;
	                                  #statSendBuffer[#statSendBufferPos] := #tempConvertedUtf8.%B2;
	                                  #statSendBufferPos += 1;
	                                ELSE  // Statement section ELSE
	                                  ;
	                              END_CASE;
	                            ELSE
	                              //When buffer full
	                              #statWillTopicEncodeState := #SUBSEQUENT_ENCODING;
	                              EXIT;
	                            END_IF;
	                          END_FOR;

	                          IF #statWillTopicPos >= LEN(#willtopic) THEN
	                            #statWillTopicEncodeState := #ENCODE_DONE;
	                          END_IF;

	                        #SUBSEQUENT_ENCODING:  // Statement section case 2 to 4
	                          FOR #tempLoopCounter := #statWillTopicPos TO LEN(#willtopic) DO
	                            "LMQTT_ConvertToUtf8"(character     := #willtopic[#tempLoopCounter],
	                                                  convertedUtf8 => #tempConvertedUtf8,
	                                                  bytesUsed     => #tempBytesUsedUtf8,
	                                                  error         => #tempErrorConvertUtf8,
	                                                  status        => #tempStatusConvertUtf8);

	                            IF #statSendBufferPos + #tempBytesUsedUtf8 <= #MAX_BUFFER_LEN_SEND THEN
	                              #statWillTopicPos += 1;
	                              CASE #tempBytesUsedUtf8 OF
	                                #UTF_1_BYTE_USED:  // Statement section case 1
	                                  #statSendBuffer[#statSendBufferPos] := #tempConvertedUtf8.%B0;
	                                  #statSendBufferPos += 1;
	                                #UTF_2_BYTE_USED:
	                                  #statSendBuffer[#statSendBufferPos] := #tempConvertedUtf8.%B0;
	                                  #statSendBufferPos += 1;
	                                  #statSendBuffer[#statSendBufferPos] := #tempConvertedUtf8.%B1;
	                                  #statSendBufferPos += 1;
	                                #UTF_3_BYTE_USED:  // Statement section case 2 to 4
	                                  #statSendBuffer[#statSendBufferPos] := #tempConvertedUtf8.%B0;
	                                  #statSendBufferPos += 1;
	                                  #statSendBuffer[#statSendBufferPos] := #tempConvertedUtf8.%B1;
	                                  #statSendBufferPos += 1;
	                                  #statSendBuffer[#statSendBufferPos] := #tempConvertedUtf8.%B2;
	                                  #statSendBufferPos += 1;
	                                ELSE  // Statement section ELSE
	                                  ;
	                              END_CASE;
	                            ELSE
	                              //When buffer full
	                              EXIT;
	                            END_IF;
	                          END_FOR;
	                          IF #statWillTopicPos >= LEN(#willtopic) THEN
	                            #statWillTopicEncodeState := #ENCODE_DONE;
	                          END_IF;

	                        ELSE  // Statement section ELSE
	                          ;
	                      END_CASE;
	                    END_IF;

	                    // Will Message
	                    // This field consists OF a two Byte length followed BY the payload FOR the Will message expressed as a sequence bytes.

	                    IF #statClientIdEncodeState = #ENCODE_DONE
	                      AND #statWillTopicEncodeState = #ENCODE_DONE
	                      AND #statSendBufferPos <= #MAX_BUFFER_LEN_SEND - #TWO_BYTE_LEN_INFO THEN
	                      //When Client Id is encoded and buffer not full
	                      CASE #statWillMessageEncodeState OF
	                        #FIRST_ENCODING:  // Statement section case 1
	                          //ADD len info into paket

	                          #tempWordForSliceAddress := UINT_TO_WORD(#statWillMessageCnt);
	                          #statSendBuffer[#statSendBufferPos] := #tempWordForSliceAddress.%B1; //MSB
	                          #statSendBufferPos += 1;
	                          #statSendBuffer[#statSendBufferPos] := #tempWordForSliceAddress.%B0; // LSB
	                          #statSendBufferPos += 1;

	                          #tempLowerWillMsgArrayBoundary := LOWER_BOUND(ARR := #willMsgPayload, DIM := #ONE_DIMENSION);

	                          IF #statWillMessageCnt > 0 THEN //will message exists
	                            FOR #tempLoopCounter := #statWillMessagePos TO UINT_TO_DINT(#statWillMessageCnt - 1) DO
	                              IF #statSendBufferPos <= #MAX_BUFFER_LEN_SEND THEN
	                                #statSendBuffer[#statSendBufferPos] := #willMsgPayload[#tempLowerWillMsgArrayBoundary + #tempLoopCounter];
	                                #statSendBufferPos += 1;
	                                //Increment when successful
	                                #statWillMessagePos += 1;
	                              ELSE
	                                //When buffer full
	                                #statWillMessageEncodeState := #SUBSEQUENT_ENCODING;
	                                EXIT;
	                              END_IF;
	                            END_FOR;
	                          END_IF;

	                          // If everything was copied successfull
	                          IF #statWillMessagePos >= #statWillMessageCnt THEN
	                            #statWillMessageEncodeState := #ENCODE_DONE;
	                          END_IF;

	                        #SUBSEQUENT_ENCODING:  // Statement section case 2 to 4
	                          #tempLowerWillMsgArrayBoundary := LOWER_BOUND(ARR := #willMsgPayload, DIM := #ONE_DIMENSION);

	                          FOR #tempLoopCounter := #statWillMessagePos TO UINT_TO_DINT(#statWillMessageCnt - 1) DO
	                            IF #statSendBufferPos <= #MAX_BUFFER_LEN_SEND THEN
	                              #statSendBuffer[#statSendBufferPos] := #willMsgPayload[#tempLowerWillMsgArrayBoundary + #tempLoopCounter];
	                              #statSendBufferPos += 1;
	                              //Increment when successful
	                              #statWillMessagePos += 1;
	                            ELSE
	                              //When Buffer Full
	                              EXIT;
	                            END_IF;
	                          END_FOR;
	                          // If everything was copied successfull
	                          IF #statWillMessagePos >= #statWillMessageCnt THEN
	                            #statWillMessageEncodeState := #ENCODE_DONE;
	                          END_IF;


	                        ELSE  // Statement section ELSE
	                          ;
	                      END_CASE;
	                    END_IF;

	                    // Username
	                    // If the Username Flag is set to 1, the Username the next field in the payload. It must be > 0 Bytes

	                    IF #statClientIdEncodeState = #ENCODE_DONE
	                      AND (#statWillTopicEncodeState = #ENCODE_DONE OR #statWillTopicEncodeState = #NOT_USED_NO_ENCODING)
	                      AND (#statWillMessageEncodeState = #ENCODE_DONE OR #statWillTopicEncodeState = #NOT_USED_NO_ENCODING)
	                      AND #statSendBufferPos <= #MAX_BUFFER_LEN_SEND - #TWO_BYTE_LEN_INFO THEN
	                      //When Will Topic and Will Message is encoded and buffer not full
	                      CASE #statUserNameEncodeState OF
	                        #FIRST_ENCODING:  // Statement section case 1
	                          //ADD len info into paket

	                          #tempWordForSliceAddress := UINT_TO_WORD(#statUsernameLenUtf8Encoded);
	                          #statSendBuffer[#statSendBufferPos] := #tempWordForSliceAddress.%B1; //MSB
	                          #statSendBufferPos += 1;
	                          #statSendBuffer[#statSendBufferPos] := #tempWordForSliceAddress.%B0; // LSB
	                          #statSendBufferPos += 1;

	                          FOR #tempLoopCounter := #statUserNamePos TO LEN(#username) DO
	                            "LMQTT_ConvertToUtf8"(character     := #username[#tempLoopCounter],
	                                                  convertedUtf8 => #tempConvertedUtf8,
	                                                  bytesUsed     => #tempBytesUsedUtf8,
	                                                  error         => #tempErrorConvertUtf8,
	                                                  status        => #tempStatusConvertUtf8);

	                            IF #statSendBufferPos + #tempBytesUsedUtf8 <= #MAX_BUFFER_LEN_SEND THEN
	                              //Increment when successful
	                              #statUserNamePos += 1;

	                              CASE #tempBytesUsedUtf8 OF
	                                #UTF_1_BYTE_USED:  // Statement section case 1
	                                  #statSendBuffer[#statSendBufferPos] := #tempConvertedUtf8.%B0;
	                                  #statSendBufferPos += 1;
	                                #UTF_2_BYTE_USED:
	                                  #statSendBuffer[#statSendBufferPos] := #tempConvertedUtf8.%B0;
	                                  #statSendBufferPos += 1;
	                                  #statSendBuffer[#statSendBufferPos] := #tempConvertedUtf8.%B1;
	                                  #statSendBufferPos += 1;
	                                #UTF_3_BYTE_USED:  // Statement section case 2 to 4
	                                  #statSendBuffer[#statSendBufferPos] := #tempConvertedUtf8.%B0;
	                                  #statSendBufferPos += 1;
	                                  #statSendBuffer[#statSendBufferPos] := #tempConvertedUtf8.%B1;
	                                  #statSendBufferPos += 1;
	                                  #statSendBuffer[#statSendBufferPos] := #tempConvertedUtf8.%B2;
	                                  #statSendBufferPos += 1;
	                                ELSE  // Statement section ELSE
	                                  ;
	                              END_CASE;
	                            ELSE
	                              //When buffer full
	                              #statUserNameEncodeState := #SUBSEQUENT_ENCODING;
	                              EXIT;
	                            END_IF;
	                          END_FOR;

	                          IF #statUserNamePos >= LEN(#username) THEN
	                            #statUserNameEncodeState := #ENCODE_DONE;
	                          END_IF;

	                        #SUBSEQUENT_ENCODING:  // Statement section case 2 to 4
	                          FOR #tempLoopCounter := #statUserNamePos TO LEN(#username) DO
	                            "LMQTT_ConvertToUtf8"(character     := #username[#tempLoopCounter],
	                                                  convertedUtf8 => #tempConvertedUtf8,
	                                                  bytesUsed     => #tempBytesUsedUtf8,
	                                                  error         => #tempErrorConvertUtf8,
	                                                  status        => #tempStatusConvertUtf8);

